   VAR_OUTPUT
      q_UDT_Status { ExternalAccessible := 'False'; ExternalVisible := 'False'; ExternalWritable := 'False'} : "UDT_SecurityCageStatus";   // Status
      qx_StartStopButtonLamp { ExternalAccessible := 'False'; ExternalVisible := 'False'; ExternalWritable := 'False'} : Bool;   // Start stop lamp button
      qx_DirectionButtonLamp { ExternalAccessible := 'False'; ExternalVisible := 'False'; ExternalWritable := 'False'} : Bool;   // Direction lamp button
      qx_ReverseDirection { ExternalAccessible := 'False'; ExternalVisible := 'False'; ExternalWritable := 'False'} : Bool;   // Signal to the system to change line direction
   END_VAR

   VAR_IN_OUT
      iq_UDT_SystemControlCommand : "UDT_SystemControlCommand";   // HMI system control structure
      iq_UDT_EquipmentControl : "UDT_EquipmentControl";   // Equipment control structure
   END_VAR

   VAR
      R_TRIG_StartStopButton {InstructionName := 'R_TRIG'; LibVersion := '1.0'; ExternalAccessible := 'False'; ExternalVisible := 'False'; ExternalWritable := 'False'; S7_SetPoint := 'False'} : R_TRIG;   // Rising edge trigger of start stop button
      R_TRIG_DirectionButton {InstructionName := 'R_TRIG'; LibVersion := '1.0'; ExternalAccessible := 'False'; ExternalVisible := 'False'; ExternalWritable := 'False'; S7_SetPoint := 'False'} : R_TRIG;   // Rising edge trigger of direction button
      sx_StartStopButtonLamp { ExternalAccessible := 'False'; ExternalVisible := 'False'; ExternalWritable := 'False'} : Bool;   // Start stop lamp button
      sx_DirectionButtonLamp { ExternalAccessible := 'False'; ExternalVisible := 'False'; ExternalWritable := 'False'} : Bool;   // Direction lamp button
      sx_Infeed { ExternalAccessible := 'False'; ExternalVisible := 'False'; ExternalWritable := 'False'} : Bool := TRUE;   // Infeed mode
      sx_Outfeed { ExternalAccessible := 'False'; ExternalVisible := 'False'; ExternalWritable := 'False'} : Bool;   // Outfeed mode
   END_VAR


BEGIN
	(*
	----------------------------------------------------------------------------------------
	|                                                                                      |
	|  Copyright  2023             Fortna Europe BV                                        |
	|  All Rights Reserved         Netherlands                                             |
	|                                                                                      |
	|                                                                                      |
	----------------------------------------------------------------------------------------

	Version history:
	Date        | Version   | Author       | Remark
	----------------------------------------------------------------------------------------
	23/11/2022  | 1.0       | S. Nikodem   | Release TIA 17 | DHL Munich 2023
	13/03/2024  | 1.1       | S. Nieswiec  | Added to new Baseline
	*)

	REGION 1 - Triggers

	    #R_TRIG_StartStopButton(CLK := #ix_StartStopButton);
	    #R_TRIG_DirectionButton(CLK := #ix_DirectionButton);

	END_REGION

	REGION 2 - Start Stop System

	    //If system is running then stop the system
	    IF #iq_UDT_EquipmentControl.Command.AutomaticOn AND #R_TRIG_StartStopButton.Q THEN

	        #iq_UDT_SystemControlCommand.Stop := True;

	    END_IF;

	    //If system is stopped then start the system
	    IF NOT #iq_UDT_EquipmentControl.Command.AutomaticOn AND #R_TRIG_StartStopButton.Q THEN

	        #iq_UDT_SystemControlCommand.Start := True;

	    END_IF;

	END_REGION

	REGION 3 - Mode

	    //Select mode
	    // The mode can be only changed when the line is stopped

	    IF NOT #iq_UDT_EquipmentControl.Command.AutomaticOn AND #R_TRIG_DirectionButton.Q THEN

	        #sx_Infeed := NOT #sx_Infeed;
	        #sx_Outfeed := NOT #sx_Outfeed;


	    END_IF;

	END_REGION

	REGION 4 - Lamp operation

	    //When the selected direction is infeed (from ground floor to security cage) the button will be solid on
	    //When the selected direction is outfeed (from the security cage to ground floor) THEN the button will be flashing at 1Hz.
	    #sx_DirectionButtonLamp := #sx_Infeed OR (#sx_Outfeed AND "mx_Clock_1Hz");


	    //When system is running then lamp will be solid on.
	    #sx_StartStopButtonLamp := #iq_UDT_EquipmentControl.Command.AutomaticOn;

	END_REGION

	REGION 5 - Status

	    #q_UDT_Status.InfeedMode := #sx_Infeed;
	    #q_UDT_Status.OutfeedMode := #sx_Outfeed;

	END_REGION

	REGION 6 - Write outputs
	    #qx_ReverseDirection := #sx_Outfeed;
	    #qx_StartStopButtonLamp := #sx_StartStopButtonLamp;
	    #qx_DirectionButtonLamp := #sx_DirectionButtonLamp;

	END_REGION

END_FUNCTION_BLOCK

FUNCTION_BLOCK "FB_RetractableRoller"
{ S7_Optimized_Access := 'TRUE' }
VERSION : 0.1
// ATTRIBUTES
// AUTO_NUMBER = True
// BLOCK_NUMBER = 100
// END_ATTRIBUTES
   VAR_INPUT
      ix_RollerError { ExternalAccessible := 'False'; ExternalVisible := 'False'; ExternalWritable := 'False'} : Bool;   // Error from roller
      ix_RollerAtHome { ExternalAccessible := 'False'; ExternalVisible := 'False'; ExternalWritable := 'False'} : Bool;   // Roller at home position
      ix_Button { ExternalAccessible := 'False'; ExternalVisible := 'False'; ExternalWritable := 'False'} : Bool;   // Switching on/off the magnet
      ix_DirectionConfig { ExternalAccessible := 'False'; ExternalVisible := 'False'; ExternalWritable := 'False'} : Bool;   // Change the direction
   END_VAR

   VAR_OUTPUT
      qx_RollerCW { ExternalAccessible := 'False'; ExternalVisible := 'False'; ExternalWritable := 'False'} : Bool;   // Forward direction
      qx_RollerCCW { ExternalAccessible := 'False'; ExternalVisible := 'False'; ExternalWritable := 'False'} : Bool;   // Revers direction
      qx_RollerRun { ExternalAccessible := 'False'; ExternalVisible := 'False'; ExternalWritable := 'False'} : Bool;   // Run Roller
      qx_Magnet { ExternalAccessible := 'False'; ExternalVisible := 'False'; ExternalWritable := 'False'} : Bool;   // On/Off Magnet
      qx_ConveyorInDieBack { ExternalAccessible := 'False'; ExternalVisible := 'False'; ExternalWritable := 'False'} : Bool;   // Active DieBack mode
      q_UDT_HMIStatus { ExternalAccessible := 'False'; ExternalVisible := 'False'; ExternalWritable := 'False'} : "UDT_RetractrableRoller_Status";   // HMI status structure
   END_VAR

   VAR_IN_OUT
      iq_UDT_ConveyorInterface : "UDT_ConveyorInterface";   // Interface structure
   END_VAR

   VAR
      s_UDT_HMI_Status { ExternalAccessible := 'False'; ExternalVisible := 'False'; ExternalWritable := 'False'; S7_SetPoint := 'False'} : "UDT_RetractrableRoller_Status";   // RetractrableRoller structure
      sx_RollerRun { ExternalAccessible := 'False'; ExternalVisible := 'False'; ExternalWritable := 'False'} : Bool;   // Roller is active
      sx_RollerCW { ExternalAccessible := 'False'; ExternalVisible := 'False'; ExternalWritable := 'False'} : Bool;   // Roller is in forward mode
      sx_RollerCCW { ExternalAccessible := 'False'; ExternalVisible := 'False'; ExternalWritable := 'False'} : Bool;   // Roller is in revers mode
      sx_Magnet { ExternalAccessible := 'False'; ExternalVisible := 'False'; ExternalWritable := 'False'} : Bool;   // Magnet is active
      sx_ConveyorInDieBack { ExternalAccessible := 'False'; ExternalVisible := 'False'; ExternalWritable := 'False'} : Bool;   // Dieback mode active
      s_UDT_CommonStatus { ExternalAccessible := 'False'; ExternalVisible := 'False'; ExternalWritable := 'False'; S7_SetPoint := 'False'} : "UDT_CommonStatus";   // Common status structure
      s_UDT_CommonStatusOld { ExternalAccessible := 'False'; ExternalVisible := 'False'; ExternalWritable := 'False'; S7_SetPoint := 'False'} : "UDT_CommonStatus";   // Common status structure
   END_VAR


BEGIN
	(*
	----------------------------------------------------------------------------------------
	|                                                                                      |
	|  Copyright  2023             FORTNA Europe BV                                        |
	|  All Rights Reserved         Netherlands                                             |
	|                                                                                      |
	----------------------------------------------------------------------------------------
	Version history:
	Date        | Version   | Author       | Remark
	----------------------------------------------------------------------------------------
	05/05/2023  | 1.0       | M. Diebel   | Release TIA 17 | DHL Munich 2023
	13/03/2024  | 1.1       | S. Nieswiec  | Added to new Baseline
	*)

	REGION 1 - Magnet handling

	    //Keep true the magnet output when the Proxy detects roller and the button is not pressed
	    #sx_Magnet := #ix_RollerAtHome AND NOT #ix_Button;

	END_REGION

	REGION 2 - Roller handling

	    // Run rollers
	    #sx_RollerRun := #ix_RollerAtHome AND (#iq_UDT_ConveyorInterface.RunFwd OR #iq_UDT_ConveyorInterface.RunRvs);

	    // Roller direction
	    IF NOT #ix_DirectionConfig
	    THEN

	        // Run rollers in forward mode
	        #sx_RollerCW := #ix_RollerAtHome AND #iq_UDT_ConveyorInterface.RunFwd AND NOT #iq_UDT_ConveyorInterface.RunRvs;

	        // Run rollers in revers mode
	        #sx_RollerCCW := #ix_RollerAtHome AND #iq_UDT_ConveyorInterface.RunRvs AND NOT #iq_UDT_ConveyorInterface.RunFwd;

	    ELSE

	        // Run rollers in forward mode
	        #sx_RollerCW := #ix_RollerAtHome AND #iq_UDT_ConveyorInterface.RunRvs AND NOT #iq_UDT_ConveyorInterface.RunFwd;

	        // Run rollers in revers mode
	        #sx_RollerCCW := #ix_RollerAtHome AND #iq_UDT_ConveyorInterface.RunFwd AND NOT #iq_UDT_ConveyorInterface.RunRvs;

	    END_IF;

	    // DieBack mode for Conveyor when roller is not at home position
	    #sx_ConveyorInDieBack := NOT #ix_RollerAtHome;

	    // Rollers is not in home position
	    #s_UDT_HMI_Status.Specific.NoHomePosition := NOT #ix_RollerAtHome;

	    // Roller reports an error
	    #s_UDT_HMI_Status.Specific.RollerError := #ix_RollerError;

	END_REGION

	REGION 3 - Status

	    //Error
	    #s_UDT_CommonStatus.Error := #s_UDT_HMI_Status.Specific.NoHomePosition;

	    //Running
	    #s_UDT_CommonStatus.Running := #sx_RollerRun AND NOT #s_UDT_HMI_Status.Specific.NoHomePosition;

	    //Stopped
	    #s_UDT_CommonStatus.Stopped := NOT #sx_RollerRun AND NOT #s_UDT_HMI_Status.Specific.NoHomePosition;

	    IF #s_UDT_CommonStatusOld <> #s_UDT_CommonStatus
	    THEN
	        // HMI status initialization
	        #s_UDT_HMI_Status.Status := 0;

	        IF #s_UDT_CommonStatus.Error
	        THEN
	            #s_UDT_HMI_Status.Status := "DB_HMIStatusConfiguration".Error;
	        END_IF;

	        IF #s_UDT_CommonStatus.Running
	        THEN
	            #s_UDT_HMI_Status.Status := "DB_HMIStatusConfiguration".Running;
	        END_IF;

	        IF #s_UDT_CommonStatus.Stopped
	        THEN
	            #s_UDT_HMI_Status.Status := "DB_HMIStatusConfiguration".Stopped;
	        END_IF;

	        #s_UDT_CommonStatusOld := #s_UDT_CommonStatus;

	    END_IF;

	END_REGION

	REGION 4 - Update outputs

	    #q_UDT_HMIStatus := #s_UDT_HMI_Status;
	    #qx_RollerCW := #sx_RollerCW;
	    #qx_RollerCCW := #sx_RollerCCW;
	    #qx_RollerRun := #sx_RollerRun;
	    #qx_Magnet := #sx_Magnet;
	    #qx_ConveyorInDieBack := #sx_ConveyorInDieBack;

	END_REGION
END_FUNCTION_BLOCK

FUNCTION_BLOCK "FB_Outfeed2States"
{ S7_Optimized_Access := 'TRUE' }
VERSION : 2.0
// ATTRIBUTES
// AUTO_NUMBER = True
// BLOCK_NUMBER = 99
// END_ATTRIBUTES
   VAR_INPUT
      i_UDT_ChuteConfiguration { ExternalAccessible := 'False'; ExternalVisible := 'False'; ExternalWritable := 'False'} : "UDT_Outfeed2StatesConfiguration";   // Chute Configuration structure
      i_UDT_AssociatedConveyorStatus { ExternalAccessible := 'False'; ExternalVisible := 'False'; ExternalWritable := 'False'} : "UDT_CommonStatus";   // Conveyor status
      ix_CapacityControlActive { ExternalAccessible := 'False'; ExternalVisible := 'False'; ExternalWritable := 'False'} : Bool;   // Chute capacity control is full
      ix_Enable { ExternalAccessible := 'False'; ExternalVisible := 'False'; ExternalWritable := 'False'} : Bool;   // TRUE when chute funcktion is enable
      ix_ConditionFull { ExternalAccessible := 'False'; ExternalVisible := 'False'; ExternalWritable := 'False'} : Bool;   // TRUE when Chute Full contidion is not blocked
      ix_ConditionHalfFull { ExternalAccessible := 'False'; ExternalVisible := 'False'; ExternalWritable := 'False'} : Bool;   // TRUE when Chute Half Full condition is not blocked
      ix_Disabled { ExternalAccessible := 'False'; ExternalVisible := 'False'; ExternalWritable := 'False'} : Bool;   // TRUE when chute is disabled
      ix_HardwareOk { ExternalAccessible := 'False'; ExternalVisible := 'False'; ExternalWritable := 'False'} : Bool;   // TRUE when chute hardware is Ok
      iudi_DelayHardwareOK { ExternalAccessible := 'False'; ExternalVisible := 'False'; ExternalWritable := 'False'} : UDInt;   // Time to delay for hardware ok signal
   END_VAR

   VAR_OUTPUT
      qx_Lamp { ExternalAccessible := 'False'; ExternalVisible := 'False'; ExternalWritable := 'False'} : Bool;   // Output Chute Lamp half full/ full
      q_UDT_HMIStatus { ExternalAccessible := 'False'; ExternalVisible := 'False'; ExternalWritable := 'False'} : "UDT_Outfeed2StatesStatus";   // HMI chute status structure
      q_UDT_Status { ExternalAccessible := 'False'; ExternalVisible := 'False'; ExternalWritable := 'False'} : "UDT_CommonStatus";   // Common chute status structure
   END_VAR

   VAR_IN_OUT
      iq_UDT_EquipmentControl : "UDT_EquipmentControl";   // Equipment control structure
      iq_ChuteExternalHandshake : "UDT_ConveyorHandshake";   // Upstream handshake structure
      iq_UDT_ConveyorHandshake : "UDT_ConveyorHandshake";
      iq_UDT_Statistics : "UDT_Outfeed2StatesStatistics";   // Statistics structure
   END_VAR

   VAR
      s_UDT_HMIStatus { ExternalAccessible := 'False'; ExternalVisible := 'False'; ExternalWritable := 'False'; S7_SetPoint := 'False'} : "UDT_Outfeed2StatesStatus";   // HMI status structure
      s_UDT_CommonStatus { ExternalAccessible := 'False'; ExternalVisible := 'False'; ExternalWritable := 'False'; S7_SetPoint := 'False'} : "UDT_CommonStatus";   // Common status structure
      s_UDT_CommonStatusOld { ExternalAccessible := 'False'; ExternalVisible := 'False'; ExternalWritable := 'False'; S7_SetPoint := 'False'} : "UDT_CommonStatus";   // Auxiliary status structure
      s_FB_HardwareOk { ExternalAccessible := 'False'; ExternalVisible := 'False'; ExternalWritable := 'False'; S7_SetPoint := 'False'} : "FB_TimerOnOffDelay";   // Timer on/off delay for hardware ok signal
      s_FB_ChuteHalfFullDetectionDelay { ExternalAccessible := 'False'; ExternalVisible := 'False'; ExternalWritable := 'False'; S7_SetPoint := 'False'} : "FB_TimerOnOffDelay";   // Timer on/off delay for chute half  full detection
      s_FB_ChuteFullDetectionDelay { ExternalAccessible := 'False'; ExternalVisible := 'False'; ExternalWritable := 'False'; S7_SetPoint := 'False'} : "FB_TimerOnOffDelay";   // Timer on/off delay for chute full detection
      s_R_TRIG_HalfFull {InstructionName := 'R_TRIG'; LibVersion := '1.0'; ExternalAccessible := 'False'; ExternalVisible := 'False'; ExternalWritable := 'False'; S7_SetPoint := 'False'} : R_TRIG;   // Rising edge trigger on chute half full signal
      s_R_TRIG_Disabled {InstructionName := 'R_TRIG'; LibVersion := '1.0'; ExternalAccessible := 'False'; ExternalVisible := 'False'; ExternalWritable := 'False'; S7_SetPoint := 'False'} : R_TRIG;   // Rising edge trigger on chute disabled signal
      s_R_TRIG_ChuteFull {InstructionName := 'R_TRIG'; LibVersion := '1.0'; ExternalAccessible := 'False'; ExternalVisible := 'False'; ExternalWritable := 'False'; S7_SetPoint := 'False'} : R_TRIG;   // Rising edge trigger on chute full signal
      s_F_TRIG_UpdateStatus {InstructionName := 'F_TRIG'; LibVersion := '1.0'; ExternalAccessible := 'False'; ExternalVisible := 'False'; ExternalWritable := 'False'; S7_SetPoint := 'False'} : F_TRIG;   // Falling edge trigger on status change
      sx_Full { ExternalAccessible := 'False'; ExternalVisible := 'False'; ExternalWritable := 'False'} : Bool;   // Full status
      sx_HalfFull { ExternalAccessible := 'False'; ExternalVisible := 'False'; ExternalWritable := 'False'} : Bool;   // Half full status
   END_VAR


BEGIN
	(*
	----------------------------------------------------------------------------------------
	|                                                                                      |
	|  Copyright  2023             FORTNA Europe BV                                        |
	|  All Rights Reserved         Netherlands                                             |
	|                                                                                      |
	----------------------------------------------------------------------------------------

	Version history:
	Date        | Version   | Author            | Remark
	----------------------------------------------------------------------------------------
	 01/03/2023 | 1.0       | R. Golonka        | Release V17 | DHL Munich
	 05/09/2023 | 1.1       | S.Theocharis      | remove the reset of restart required
	 05/09/2023 | 1.2       | M.Diebel          | Initilization, s_UDT_CommonStatus.Stopped set on true
	 06/09/2023 | 1.3       | M.Diebel          | Rewrite reset energy save from external handshake to conveyor handshake
	 12/09/2023 | 2.0       | M.Diebel          | Set status "stopped" when chute is disable
	 13/03/2024 | 2.1       | S. Nieswiec       | Added to new Baseline


	 *)


	REGION 1 - Inicialization
	    //Reset HMI status and Common status and exit
	    IF NOT #ix_Enable THEN
	        #s_UDT_HMIStatus.Specific.ChuteFull := 0;
	        #s_UDT_HMIStatus.Specific.ChuteHalfFull := 0;
	        #s_UDT_HMIStatus.Specific.ChuteDisabled := 0;
	        #s_UDT_CommonStatus.SafetyStop := 0;
	        #s_UDT_CommonStatus.AutoON := 0;
	        #s_UDT_CommonStatus.Stopped := TRUE;
	        #s_UDT_HMIStatus.Status := "DB_HMIStatusConfiguration".Stopped;
	        #q_UDT_HMIStatus := #s_UDT_HMIStatus;
	        #q_UDT_Status := #s_UDT_CommonStatus;
	        #iq_UDT_EquipmentControl.Report := #s_UDT_CommonStatus;
	        #qx_Lamp := 0;
	        #iq_UDT_ConveyorHandshake.RTS := 0;
	        #iq_ChuteExternalHandshake.RTR := 0;

	        RETURN;
	    END_IF;
	END_REGION

	REGION 2 - Timers

	    // Chute full detection timer
	    #s_FB_ChuteFullDetectionDelay(iudi_OnDelayTime := #i_UDT_ChuteConfiguration.FullDetectionTime,
	                                  iudi_OffDelayTime := #i_UDT_ChuteConfiguration.FullReleaseTime,
	                                  ix_SignalToDelay := NOT #ix_ConditionFull,
	                                  qx_DelayedSignal => #sx_Full);

	    // Chute half full detection timer
	    #s_FB_ChuteHalfFullDetectionDelay(iudi_OnDelayTime := #i_UDT_ChuteConfiguration.HalfFullDetectionTime,
	                                      iudi_OffDelayTime := #i_UDT_ChuteConfiguration.HalfFullReleaseTime,
	                                      ix_SignalToDelay := NOT #ix_ConditionHalfFull,
	                                      qx_DelayedSignal => #sx_HalfFull);

	    // Hardware ok signal delay
	    #s_FB_HardwareOk(iudi_OnDelayTime := #iudi_DelayHardwareOK,
	                     ix_SignalToDelay := #ix_HardwareOk);


	END_REGION

	REGION 3 - Stop upstream conveyor

	    // Stop upstream conveyor when chute is full or disabled
	    #iq_ChuteExternalHandshake.RTR := NOT #sx_Full AND NOT #ix_CapacityControlActive AND NOT #ix_Disabled AND #s_FB_HardwareOk.qx_DelayedSignal AND #iq_UDT_EquipmentControl.Report.AutoON;

	END_REGION

	REGION 4 - Start next conveyor

	    // Start conveyor when upstream conveyor is running
	    #iq_UDT_ConveyorHandshake.RTS := #iq_ChuteExternalHandshake.RTR;
	    #iq_UDT_ConveyorHandshake.ResetEnergySave := #iq_ChuteExternalHandshake.ResetEnergySave;
	END_REGION


	REGION 5 - Update output

	    // Update the outputs
	    #qx_Lamp := (#sx_Full OR (#sx_HalfFull AND "DB_Memory".Clock_1Hz));

	END_REGION

	REGION 6 - Status

	    // Update chute full specific status
	    #s_UDT_HMIStatus.Specific.ChuteFull := #sx_Full AND #s_FB_HardwareOk.qx_DelayedSignal;

	    // Update chute half full specific status
	    #s_UDT_HMIStatus.Specific.ChuteHalfFull := #sx_HalfFull AND #s_FB_HardwareOk.qx_DelayedSignal;

	    //Update chute disabled specific status
	    #s_UDT_HMIStatus.Specific.ChuteDisabled := #ix_Disabled AND #s_FB_HardwareOk.qx_DelayedSignal;


	    // Update common safety stop
	    #s_UDT_CommonStatus.SafetyStop := #i_UDT_AssociatedConveyorStatus.SafetyStop;

	    // Update common automatic on
	    #s_UDT_CommonStatus.AutoON := #i_UDT_AssociatedConveyorStatus.AutoON;

	    // Update common stopped
	    #s_UDT_CommonStatus.Stopped := #i_UDT_AssociatedConveyorStatus.Stopped;


	    // Update HMI status number for chute disabled
	    IF #s_UDT_HMIStatus.Specific.ChuteDisabled AND NOT #s_UDT_CommonStatus.SafetyStop
	    THEN
	        #s_UDT_HMIStatus.Status := "DB_HMIStatusConfiguration".DisableByManagement;
	    END_IF;

	    // Update HMI status number for chute half full
	    IF #s_UDT_HMIStatus.Specific.ChuteHalfFull AND NOT #s_UDT_CommonStatus.SafetyStop
	    THEN
	        #s_UDT_HMIStatus.Status := "DB_HMIStatusConfiguration".ChuteHalfFull;
	    END_IF;

	    // Update HMI status number for chute full
	    IF #s_UDT_HMIStatus.Specific.ChuteFull AND NOT #s_UDT_CommonStatus.SafetyStop
	    THEN
	        #s_UDT_HMIStatus.Status := "DB_HMIStatusConfiguration".ChuteFull;
	    END_IF;


	    // Collecting F_TRIG on chute full, chute half full or chute disabled status to update common status
	    #s_F_TRIG_UpdateStatus(CLK := #s_UDT_HMIStatus.Specific.ChuteFull
	                           OR #s_UDT_HMIStatus.Specific.ChuteDisabled
	                           OR #s_UDT_HMIStatus.Specific.ChuteHalfFull);

	    // HMI status number calculation
	    IF #s_UDT_CommonStatusOld <> #s_UDT_CommonStatus OR #s_F_TRIG_UpdateStatus.Q
	    THEN

	        // Update auto on status number
	        IF #s_UDT_CommonStatus.AutoON
	        THEN
	            #s_UDT_HMIStatus.Status := "DB_HMIStatusConfiguration".AutoON;

	        END_IF;

	        IF #s_UDT_CommonStatus.Stopped
	        THEN
	            #s_UDT_HMIStatus.Status := "DB_HMIStatusConfiguration".Stopped;

	        END_IF;

	        IF #s_UDT_CommonStatus.SafetyStop
	        THEN
	            #s_UDT_HMIStatus.Status := "DB_HMIStatusConfiguration".SafetyStop;

	        END_IF;

	        // Copy common status structure to the old common status structure
	        #s_UDT_CommonStatusOld := #s_UDT_CommonStatus;
	        #q_UDT_Status := #s_UDT_CommonStatus;

	    END_IF;

	    #q_UDT_HMIStatus := #s_UDT_HMIStatus;

	END_REGION

	REGION 7 - Statistics

	    // Chute full R_TRIG for statistics purpose
	    #s_R_TRIG_ChuteFull(CLK := #s_UDT_HMIStatus.Specific.ChuteFull);

	    // Chute full statistics
	    IF #s_UDT_HMIStatus.Specific.ChuteFull
	        OR #iq_UDT_EquipmentControl.Command.ResetData
	    THEN
	        "FC_Statistics"(ix_Reset := #iq_UDT_EquipmentControl.Command.ResetData,
	                        ix_Activate := #s_UDT_HMIStatus.Specific.ChuteFull,
	                        ix_RTrigActivate := #s_R_TRIG_ChuteFull.Q,
	                        iqUDT_Statistics := #iq_UDT_Statistics.ChuteFull);

	    END_IF;

	    // Chute disabled R_TRIG for statistics purpose
	    #s_R_TRIG_Disabled(CLK := #s_UDT_HMIStatus.Specific.ChuteDisabled);

	    // Chute disabled statistics
	    IF #s_UDT_HMIStatus.Specific.ChuteDisabled
	        OR #iq_UDT_EquipmentControl.Command.ResetData
	    THEN
	        "FC_Statistics"(ix_Reset := #iq_UDT_EquipmentControl.Command.ResetData,
	                        ix_Activate := #s_UDT_HMIStatus.Specific.ChuteDisabled,
	                        ix_RTrigActivate := #s_R_TRIG_Disabled.Q,
	                        iqUDT_Statistics := #iq_UDT_Statistics.ChuteDisabled);

	    END_IF;

	    // Chute half full R_TRIG for statistics purpose
	    #s_R_TRIG_HalfFull(CLK := #s_UDT_HMIStatus.Specific.ChuteHalfFull);

	    // Chute half full statistics
	    IF #s_UDT_HMIStatus.Specific.ChuteHalfFull
	        OR #iq_UDT_EquipmentControl.Command.ResetData
	    THEN

	        "FC_Statistics"(ix_Reset := #iq_UDT_EquipmentControl.Command.ResetData,
	                        ix_Activate := #s_UDT_HMIStatus.Specific.ChuteHalfFull,
	                        ix_RTrigActivate := #s_R_TRIG_HalfFull.Q,
	                        iqUDT_Statistics := #iq_UDT_Statistics.ChuteHalfFull);

	    END_IF;

	END_REGION

	REGION 8 - Equipment Report

	    "FC_EquipmentReport"(iUDT_Status := #s_UDT_CommonStatus,
	                         iqUDT_Control := #iq_UDT_EquipmentControl);

	END_REGION
END_FUNCTION_BLOCK

FUNCTION_BLOCK "FB_InchingBulkV2"
{ S7_Optimized_Access := 'TRUE' }
VERSION : 0.1
// ATTRIBUTES
// AUTO_NUMBER = True
// BLOCK_NUMBER = 97
// END_ATTRIBUTES
   VAR_INPUT
      ix_PECUp { ExternalAccessible := 'False'; ExternalVisible := 'False'; ExternalWritable := 'False'} : Bool;   // PEC Sum signal from upstream conveyor
      ix_LongParcelDetection { ExternalAccessible := 'False'; ExternalVisible := 'False'; ExternalWritable := 'False'} : Bool;   // Long parcel detection PEC's
      ix_InchingActive { ExternalAccessible := 'False'; ExternalVisible := 'False'; ExternalWritable := 'False'} : Bool;   // If TRUE inching is activate
      ix_InchingLineHealthy { ExternalAccessible := 'False'; ExternalVisible := 'False'; ExternalWritable := 'False'} : Bool;
      ix_ClearCommand { ExternalAccessible := 'False'; ExternalVisible := 'False'; ExternalWritable := 'False'} : Bool;   // Command to clear full status
      ix_DownstreamFull { ExternalAccessible := 'False'; ExternalVisible := 'False'; ExternalWritable := 'False'} : Bool;   // TRUE if downstream conveyors are full
      ii_OnDelayGap { ExternalAccessible := 'False'; ExternalVisible := 'False'; ExternalWritable := 'False'} : DInt;   // Distance to conveyor release [mm]
      ii_InchingGap { ExternalAccessible := 'False'; ExternalVisible := 'False'; ExternalWritable := 'False'} : DInt;   // Inching distance [mm]
      ii_Displacement_Upstream { ExternalAccessible := 'False'; ExternalVisible := 'False'; ExternalWritable := 'False'} : Int;   // Upstream conveyor displacement
      ii_Displacement { ExternalAccessible := 'False'; ExternalVisible := 'False'; ExternalWritable := 'False'} : Int;   // Inching conveyor displacement
      iudt_ConveyorInterface { ExternalAccessible := 'False'; ExternalVisible := 'False'; ExternalWritable := 'False'} : "UDT_ConveyorInterface";
   END_VAR

   VAR_OUTPUT
      qx_ExternalRequestHold { ExternalAccessible := 'False'; ExternalVisible := 'False'; ExternalWritable := 'False'} : Bool;   // External output to request conveyor hold
      qx_Full { ExternalAccessible := 'False'; ExternalVisible := 'False'; ExternalWritable := 'False'} : Bool;   // Inching conveyor is full status
   END_VAR

   VAR
      s_FB_TimerOnOffDelay_LongParcelDetection { ExternalAccessible := 'False'; ExternalVisible := 'False'; ExternalWritable := 'False'; S7_SetPoint := 'False'} : "FB_TimerOnOffDelay";
      F_TRIG_PECEoSUp {InstructionName := 'F_TRIG'; LibVersion := '1.0'; ExternalAccessible := 'False'; ExternalVisible := 'False'; ExternalWritable := 'False'; S7_SetPoint := 'False'} : F_TRIG;   // Falling edge trigger PEC EoS
      si_ActualInchingGap { ExternalAccessible := 'False'; ExternalVisible := 'False'; ExternalWritable := 'False'} : Int;   // Distance to request hold
      si_ActualOnGap { ExternalAccessible := 'False'; ExternalVisible := 'False'; ExternalWritable := 'False'} : Int;   // Distance to conveyor release
      sx_StartRelease { ExternalAccessible := 'False'; ExternalVisible := 'False'; ExternalWritable := 'False'} : Bool;   // Conveyor release
      sx_ConveyorFull { ExternalAccessible := 'False'; ExternalVisible := 'False'; ExternalWritable := 'False'} : Bool;
      s_Status { ExternalAccessible := 'False'; ExternalVisible := 'False'; ExternalWritable := 'False'; S7_SetPoint := 'False'} : "UDT_InchingStatus";
      s_StatusOld { ExternalAccessible := 'False'; ExternalVisible := 'False'; ExternalWritable := 'False'; S7_SetPoint := 'False'} : "UDT_InchingStatus";
      sx_InchingActive { ExternalAccessible := 'False'; ExternalVisible := 'False'; ExternalWritable := 'False'} : Bool;
   END_VAR


BEGIN
	(*
	----------------------------------------------------------------------------------------
	|                                                                                      |
	|  Copyright  2019             MHS                                                     |
	|  All Rights Rese9ved         Larenweg 90                                             |
	|                              5234 KC 's-Hertogenbosch,                               |
	|                              Netherlands                                             |
	|                                                                                      |
	----------------------------------------------------------------------------------------

	Version history:
	Date        | Version   | Author        | Remark
	----------------------------------------------------------------------------------------
	01/04/2021 | 1.0       | M.Kocot      | first release TIA 16
	08/04/2021 | 1.1       | H.Rutkwoski  | Added status full
	14/08/2021 | 1.2       | M. Jager     | Reset sx_full when inching is not active
	26/07/2023 | 1.3       | S.Nikodem    | Absolut displacement value
	13/09/2023 | 1.4       | M.Diebel     | Activate inching if PEC is clear
	14/09/2023 | 1.5       | M.Diebel     | Hold line when downstream conveyors are full
	06/02/2024 | 1.6       | L.Klar       | Long parcel detection
	13/03/2024 | 1.7       | S. Nieswiec  | Changed name to V2
	*)

	REGION 1 - Triggers

	    // Falling edge trigger PEC EoS.
	    #F_TRIG_PECEoSUp(CLK := #ix_PECUp);

	END_REGION

	REGION 2 - TTimers

	    #s_FB_TimerOnOffDelay_LongParcelDetection(iudi_OffDelayTime := 100,
	                                              ix_SignalToDelay := #ix_LongParcelDetection);

	END_REGION

	REGION 3 - Inching
	    // Statement section REGION

	    //Activate inching if PEC is clear
	    #sx_InchingActive := #ix_InchingActive AND (#sx_InchingActive OR #ix_PECUp);



	    IF ((#F_TRIG_PECEoSUp.Q OR NOT #s_FB_TimerOnOffDelay_LongParcelDetection.qx_DelayedSignal) AND #sx_InchingActive)
	        // OR( RisingeEdge of Ix_InchigActive AND NOT IX_PECup )
	    THEN
	        #si_ActualOnGap := DINT_TO_INT(#ii_OnDelayGap / 10);
	        #si_ActualInchingGap := DINT_TO_INT(#ii_InchingGap / 10);

	    END_IF;

	    IF #si_ActualOnGap > 0 THEN

	        #si_ActualOnGap := #si_ActualOnGap - ABS(#ii_Displacement_Upstream);

	    END_IF;

	    IF #ix_PECUp AND #si_ActualInchingGap > 0 THEN
	        #si_ActualInchingGap := #si_ActualInchingGap - ABS(#ii_Displacement);
	    END_IF;

	    IF #si_ActualOnGap <= 0
	        //  OR #sx_StartRelease
	    THEN
	        #sx_StartRelease := TRUE;
	    END_IF;

	    IF (#si_ActualInchingGap <= 0)
	    THEN
	        #sx_StartRelease := FALSE;
	    END_IF;

	    #qx_ExternalRequestHold := (((NOT #sx_StartRelease OR NOT #ix_InchingLineHealthy) OR #ix_DownstreamFull) AND #sx_InchingActive);

	END_REGION

	REGION 4 - Internal status - conveyor full

	    // Set conveyor status to full when:
	    IF #sx_InchingActive                     // inching is active
	        AND #ix_DownstreamFull               // downstream is full
	        AND NOT #ix_ClearCommand             // there is no clear command active
	    THEN
	        #sx_ConveyorFull := TRUE;
	    END_IF;

	    // Set conveyor status to NOT full when:
	    IF (#sx_InchingActive                   // Inching is active
	        AND #ix_ClearCommand                // clear command is active
	        AND NOT #ix_DownstreamFull)         // downstream is NOT full)
	        OR NOT #sx_InchingActive            // OR Inching isnt active
	    THEN
	        #sx_ConveyorFull := FALSE;
	    END_IF;

	END_REGION

	REGION 5 - Status

	    // Convsyor is full status
	    #s_Status.Full := #sx_ConveyorFull;

	    #s_Status.Active := #sx_InchingActive;

	    // Status update on change.
	    IF #s_StatusOld <> #s_Status
	    THEN
	        #qx_Full := #s_Status.Full;
	        #s_StatusOld := #s_Status;
	    END_IF;

	END_REGION
END_FUNCTION_BLOCK

FUNCTION_BLOCK "FB_SNCY_Infeed"
{ S7_Optimized_Access := 'TRUE' }
VERSION : 0.1
// ATTRIBUTES
// AUTO_NUMBER = True
// BLOCK_NUMBER = 242
// END_ATTRIBUTES
   VAR_INPUT
      ix_KneeButton { ExternalAccessible := 'False'; ExternalVisible := 'False'; ExternalWritable := 'False'} : Bool;   // Signal from knee button
      ix_ResetButton { ExternalAccessible := 'False'; ExternalVisible := 'False'; ExternalWritable := 'False'} : Bool;   // Signal from reset button
      ix_PEC_EoS { ExternalAccessible := 'False'; ExternalVisible := 'False'; ExternalWritable := 'False'} : Bool;   // Sensor at end of conveyor
      i_UDT_PECUpdateConfiguration { ExternalAccessible := 'False'; ExternalVisible := 'False'; ExternalWritable := 'False'} : "UDT_PECUpdateConfiguration";   // PEC update configuration
      idtl_ActualTime {InstructionName := 'DTL'; LibVersion := '1.0'; ExternalAccessible := 'False'; ExternalVisible := 'False'; ExternalWritable := 'False'} : DTL;   // Actual date and time in DTL
   END_VAR

   VAR_OUTPUT
      qx_ConveyorHold { ExternalAccessible := 'False'; ExternalVisible := 'False'; ExternalWritable := 'False'} : Bool;   // Hold command for conveyor
      qx_WhiteLamp { ExternalAccessible := 'False'; ExternalVisible := 'False'; ExternalWritable := 'False'} : Bool;   // White signal lamp
      qx_BlueLamp { ExternalAccessible := 'False'; ExternalVisible := 'False'; ExternalWritable := 'False'} : Bool;   // Blue signal lamp
   END_VAR

   VAR_IN_OUT
      iqa_TrackingData : Array[*] of Int;   // Conveyor tracking data
      iq_UDT_FifoHeaderMFCMessage : "UDT_FifoHeader";   // FIFO header of generated messages
      iqs_FifoDataMFCMessage : Array[*] of "UDT_MessageV2";   // FIFO data Buffer of generated messages
      iqdi_MessageSequenceNumber { ExternalAccessible := 'False'; ExternalVisible := 'False'; ExternalWritable := 'False'} : Int;   // MFC Sort - Message number
      iqs_MFCNewObjectID : String;   // New Object ID number received from MFC
      is_MFCRejectObjectID : String;   // Number received from MFC with the order to reject the package (ObjectID)
   END_VAR

   VAR
      s_FB_MFC_Sort_VIDResponse_ASCII { ExternalAccessible := 'False'; ExternalVisible := 'False'; ExternalWritable := 'False'; S7_SetPoint := 'False'} : "FB_MFC_Sort_VIDResponse_ASCII";   // VID message generator
      F_TRIG_PEC_EoS {InstructionName := 'F_TRIG'; LibVersion := '1.0'; ExternalAccessible := 'False'; ExternalVisible := 'False'; ExternalWritable := 'False'; S7_SetPoint := 'False'} : F_TRIG;   // Rising edge for photo eye
      sx_WaitForObjectID { ExternalAccessible := 'False'; ExternalVisible := 'False'; ExternalWritable := 'False'} : Bool;   // True - Parcel is in position, wait for information from MFC
      sx_WaitForDestination { ExternalAccessible := 'False'; ExternalVisible := 'False'; ExternalWritable := 'False'} : Bool;   // True - Parcel is in position, wait for information from MFC
      sx_WaitForParcel { ExternalAccessible := 'False'; ExternalVisible := 'False'; ExternalWritable := 'False'} : Bool;   // True - Information from MFC received , wait for parcel
      sx_ParcelReject { ExternalAccessible := 'False'; ExternalVisible := 'False'; ExternalWritable := 'False'} : Bool;   // True - The parcel is rejected by the MFC system
   END_VAR

   VAR_TEMP
      tudi_MFCRejectObjectID : UDInt;   // MFC Reject Object ID
   END_VAR


BEGIN
	(*
	----------------------------------------------------------------------------------------
	|                                                                                      |
	|  Copyright  2023             FORTNA Europe BV                                        |
	|  All Rights Reserved         Netherlands                                             |
	|                                                                                      |
	----------------------------------------------------------------------------------------
	Version history:
	Date        | Version   | Author       | Remark
	----------------------------------------------------------------------------------------
	28/06/2023  | 1.0       | S. Nikodem   | Release TIA 17 | DHL Munich 2023
	13/09/2023  | 1.1       | S. Nikodem   | Update interface
	13/03/2024  | 1.2       | S. Nieswiec  | Added to new baseline, block needs uptade after munich is finished
	*)

	REGION 1 - Triggers

	    // Rising edge - Parcel detected
	    #F_TRIG_PEC_EoS(CLK := #ix_PEC_EoS);

	END_REGION

	REGION 2 - Buttons

	    //Knee button
	    IF #ix_KneeButton AND #ix_PEC_EoS THEN

	        #sx_WaitForParcel := True;

	    END_IF;

	    //Reset button
	    //Reset after removing the package.
	    IF #ix_ResetButton AND #ix_PEC_EoS AND #sx_ParcelReject THEN
	        #sx_ParcelReject := False;
	    END_IF;

	END_REGION

	REGION 3 - Data

	    REGION 3.1 - Object ID

	        IF (#iqa_TrackingData[#i_UDT_PECUpdateConfiguration.Distance] > 0) THEN

	            //Match GIN with Object ID
	            IF NOT #ix_PEC_EoS                                                          // Parcel on the sensor
	                AND NOT "DB_GIN".GIN[#iqa_TrackingData[#i_UDT_PECUpdateConfiguration.Distance]].DHL.MFCMessage.Received.TemporaryParcelIdentifier  //The message for this GIN has not yet been received.
	                AND NOT (#iqs_MFCNewObjectID = '0')                                             // New Object ID
	            THEN

	                //Copy data from MFC
	                "DB_GIN".GIN[#iqa_TrackingData[#i_UDT_PECUpdateConfiguration.Distance]].DHL.ObjectID := #iqs_MFCNewObjectID;

	                //Temporary Parcel Identifier message with Object ID received
	                "DB_GIN".GIN[#iqa_TrackingData[#i_UDT_PECUpdateConfiguration.Distance]].DHL.MFCMessage.Received.TemporaryParcelIdentifier := True;
	                "DB_GIN".GIN[#iqa_TrackingData[#i_UDT_PECUpdateConfiguration.Distance]].General.Identification.GoodRead := True;

	                // Generate VID
	                #s_FB_MFC_Sort_VIDResponse_ASCII(is_ObjectID := #iqs_MFCNewObjectID,
	                                                 i_ActualTimeDTL := #idtl_ActualTime,
	                                                 iq_UDT_FifoHeader := #iq_UDT_FifoHeaderMFCMessage,
	                                                 iqs_FifoData := #iqs_FifoDataMFCMessage,
	                                                 iqdi_MessageSequenceNumber := #iqdi_MessageSequenceNumber);

	                //VID Response message generated
	                "DB_GIN".GIN[#iqa_TrackingData[#i_UDT_PECUpdateConfiguration.Distance]].DHL.MFCMessage.Sent.VIDResponse := True;

	                //Reset data in DB_MFC
	                #iqs_MFCNewObjectID := '0';

	                //Reset value
	                #sx_WaitForObjectID := False;

	            END_IF;

	        END_IF;


	    END_REGION

	    REGION 3.2 -Destination

	        IF (#iqa_TrackingData[#i_UDT_PECUpdateConfiguration.Distance] > 0) THEN

	            IF NOT #ix_PEC_EoS                                                              // Parcel on the sensor
	                AND NOT #sx_WaitForObjectID                                                 // Object ID received
	                AND "DB_GIN".GIN[#iqa_TrackingData[#i_UDT_PECUpdateConfiguration.Distance]].DHL.MFCMessage.Received.Destination                    //The message for this GIN has been received.
	            THEN

	                //Reset value
	                #sx_WaitForDestination := False;

	            END_IF;

	        END_IF;

	    END_REGION

	    REGION 3.3 - Parcel Reject

	        #tudi_MFCRejectObjectID := STRING_TO_UDINT(#is_MFCRejectObjectID);

	        IF (#iqa_TrackingData[#i_UDT_PECUpdateConfiguration.Distance] > 0) THEN

	            IF NOT #ix_PEC_EoS                                                          // Parcel on the sensor
	                AND NOT #sx_WaitForObjectID                                             // Object ID received
	                AND #tudi_MFCRejectObjectID > 0                       // New destination message from MFC reveived
	                AND ("DB_GIN".GIN[#iqa_TrackingData[#i_UDT_PECUpdateConfiguration.Distance]].DHL.ObjectID = #is_MFCRejectObjectID)
	                AND NOT "DB_GIN".GIN[#iqa_TrackingData[#i_UDT_PECUpdateConfiguration.Distance]].DHL.MFCMessage.Received.RejectParcel //The message for this GIN has not yet been received.
	            THEN

	                //Reject parcel received
	                "DB_GIN".GIN[#iqa_TrackingData[#i_UDT_PECUpdateConfiguration.Distance]].DHL.MFCMessage.Received.RejectParcel := True;

	                //Reset data in DB_MFC
	                #is_MFCRejectObjectID := '0';

	                //Reset value
	                #sx_WaitForDestination := False;

	                //Set value
	                #sx_ParcelReject := True;

	            END_IF;

	        END_IF;

	    END_REGION

	    //Hold conveyor if parcel is detected
	    IF #F_TRIG_PEC_EoS.Q THEN
	        #sx_WaitForObjectID := True;
	        #sx_WaitForDestination := True;
	        #sx_WaitForParcel := FALSE;
	    END_IF;

	    //Data received wait for parcel
	    IF NOT (#iqs_MFCNewObjectID = '0') THEN
	        #sx_WaitForParcel := True;
	    END_IF;

	    //Hold
	    #qx_ConveyorHold := NOT #sx_WaitForParcel AND (#sx_WaitForDestination OR #sx_ParcelReject);

	END_REGION

	REGION 4 - Lamp handling

	    //White lamp
	    //1 hz - Parcel on the sensor, waiting for data from MFC
	    //On - Waiting for a package
	    #qx_WhiteLamp := NOT #sx_ParcelReject AND (NOT #ix_PEC_EoS OR (#sx_WaitForObjectID AND "DB_Memory".Clock_1Hz));

	    //Blue lamp
	    //1 hz - Parcel reject
	    #qx_BlueLamp := #sx_ParcelReject AND "DB_Memory".Clock_1Hz;

	END_REGION
END_FUNCTION_BLOCK

FUNCTION_BLOCK "FB_EuchnerLockV2"
{ S7_Optimized_Access := 'TRUE' }
VERSION : 0.1
// ATTRIBUTES
// AUTO_NUMBER = True
// BLOCK_NUMBER = 96
// END_ATTRIBUTES
   VAR_INPUT
      ix_ButtonReset { ExternalAccessible := 'False'; ExternalVisible := 'False'; ExternalWritable := 'False'} : Bool;   // Reset button
      ix_ButtonRequest { ExternalAccessible := 'False'; ExternalVisible := 'False'; ExternalWritable := 'False'} : Bool;   // Request open button
      ix_IdCardAccessGranted { ExternalAccessible := 'False'; ExternalVisible := 'False'; ExternalWritable := 'False'} : Bool;   // Feedback from DHL- ID card ok - access granted
      ix_DoorClosed { ExternalAccessible := 'False'; ExternalVisible := 'False'; ExternalWritable := 'False'} : Bool;   // Feedback from lock - door is closed
      ix_BoltTongueClosed { ExternalAccessible := 'False'; ExternalVisible := 'False'; ExternalWritable := 'False'} : Bool;   // Feedback from lock - bolt tongue closed
      ix_SafelyLoced { ExternalAccessible := 'False'; ExternalVisible := 'False'; ExternalWritable := 'False'} : Bool;   // Feedback from lock - Safely locked
      ix_InternalErrorReset { ExternalAccessible := 'False'; ExternalVisible := 'False'; ExternalWritable := 'False'} : Bool;   // Internal error reset command from system control
      ix_LockFault { ExternalAccessible := 'False'; ExternalVisible := 'False'; ExternalWritable := 'False'} : Bool;   // Lock has an internal fault
      ix_SystemStopped { ExternalAccessible := 'False'; ExternalVisible := 'False'; ExternalWritable := 'False'} : Bool;   // Feedback from system - System is stopped
      ix_SafetyLockOK { ExternalAccessible := 'False'; ExternalVisible := 'False'; ExternalWritable := 'False'} : Bool;   // Safety lock status OK
      ix_SafetyLockAckReq { ExternalAccessible := 'False'; ExternalVisible := 'False'; ExternalWritable := 'False'} : Bool;   // Safety lock need acknowledgement
      ii_NumberOfLEDs { ExternalAccessible := 'False'; ExternalVisible := 'False'; ExternalWritable := 'False'} : Int;   // Number of programmable LEDs on lock
   END_VAR

   VAR_OUTPUT
      qx_StopSystem { ExternalAccessible := 'False'; ExternalVisible := 'False'; ExternalWritable := 'False'} : Bool;   // Signal to stop the system
      qx_ResetButtonLed { ExternalAccessible := 'False'; ExternalVisible := 'False'; ExternalWritable := 'False'} : Bool;   // Reset button lamp
      qx_RequestButtonLed { ExternalAccessible := 'False'; ExternalVisible := 'False'; ExternalWritable := 'False'} : Bool;   // Request button lamp
      qx_FaultReset { ExternalAccessible := 'False'; ExternalVisible := 'False'; ExternalWritable := 'False'} : Bool;   // Reset internal lock fault
      qx_SafetyReset { ExternalAccessible := 'False'; ExternalVisible := 'False'; ExternalWritable := 'False'} : Bool;   // Safety reset command after authorization
      qx_ReleaseLock { ExternalAccessible := 'False'; ExternalVisible := 'False'; ExternalWritable := 'False'} : Bool;   // Signal to safety logic to release lock
      q_UDT_Status { ExternalAccessible := 'False'; ExternalVisible := 'False'; ExternalWritable := 'False'} : "UDT_EuchnerLockStatusV2";   // Status structure
   END_VAR

   VAR
      s_R_TRIG_RequestButton {InstructionName := 'R_TRIG'; LibVersion := '1.0'; ExternalAccessible := 'False'; ExternalVisible := 'False'; ExternalWritable := 'False'; S7_SetPoint := 'False'} : R_TRIG;   // Rising edge trigger from reqest button
      s_F_TRIG_BoltTongueClosed {InstructionName := 'F_TRIG'; LibVersion := '1.0'; ExternalAccessible := 'False'; ExternalVisible := 'False'; ExternalWritable := 'False'; S7_SetPoint := 'False'} : F_TRIG;   // Falling edge trigger from bolt tongue
      s_F_TRIG_ReleaseLock {InstructionName := 'F_TRIG'; LibVersion := '1.0'; ExternalAccessible := 'False'; ExternalVisible := 'False'; ExternalWritable := 'False'; S7_SetPoint := 'False'} : F_TRIG;   // Falling edge trigger from release lock
      s_FB_TimerOnOffDelay { ExternalAccessible := 'False'; ExternalVisible := 'False'; ExternalWritable := 'False'; S7_SetPoint := 'False'} : "FB_TimerOnOffDelay";   // Function block to generate on signal delay - emergency request button
      s_FB_TimerOnOffDelay_ResetDelay { ExternalAccessible := 'False'; ExternalVisible := 'False'; ExternalWritable := 'False'; S7_SetPoint := 'False'} : "FB_TimerOnOffDelay";
      sx_Request { ExternalAccessible := 'False'; ExternalVisible := 'False'; ExternalWritable := 'False'} : Bool;   // Request to open the door
      sx_ReqMissingAccessRights { ExternalAccessible := 'False'; ExternalVisible := 'False'; ExternalWritable := 'False'} : Bool;   // Button access request triggered without permission from DHL
      sx_ResetMissingAccessRights { ExternalAccessible := 'False'; ExternalVisible := 'False'; ExternalWritable := 'False'} : Bool;   // Button Reset triggered without permission from DHL
      sx_DoorOpenedWithoutReq { ExternalAccessible := 'False'; ExternalVisible := 'False'; ExternalWritable := 'False'} : Bool;   // Doors were opened without request and permission
   END_VAR

   VAR CONSTANT
      c_Time : UDInt := 10000;
   END_VAR


BEGIN

	(*
	----------------------------------------------------------------------------------------
	|                                                                                      |
	|  Copyright  2023             FORTNA Europe BV                                        |
	|  All Rights Reserved         Netherlands                                             |
	|                                                                                      |
	----------------------------------------------------------------------------------------

	Version history:
	Date        | Version   | Author       | Remark
	----------------------------------------------------------------------------------------
	11/03/2022  | 0.1       | S.Nikodem    | first release MHS TIA 15.1
	24/08/2022  | 0.2       | K. Pokorski  | Change to Lock with key switch and only one LED
	11/10/2023  | 0.3       | M.Diebel     | first release Fortna TIA 17
	30/01/2024  | 0.4       | A. Bunzel    | Add logic for ID cards from DHL
	13/03/2024  | 0.5       | S. Nieswiec  | Changed name to V2
	*)

	REGION 1 - Request open

	    //Button
	    //Rising edge trigger
	    #s_R_TRIG_RequestButton(CLK := #ix_ButtonRequest);

	    // Flip-flop
	    IF #s_R_TRIG_RequestButton.Q AND #ix_IdCardAccessGranted THEN

	        IF #sx_Request THEN
	            #sx_Request := FALSE;
	        ELSE
	            #sx_Request := TRUE;
	        END_IF;

	    END_IF;

	    // Reset Flip-Flop
	    IF NOT #ix_BoltTongueClosed THEN
	        #sx_Request := FALSE;
	    END_IF;

	    //Stop system
	    #qx_StopSystem := #sx_Request;

	    //If system is stopped and is safe then open lock
	    #qx_ReleaseLock := (#sx_Request AND #ix_SystemStopped);

	END_REGION

	REGION 2 - Lamp controlling


	    CASE #ii_NumberOfLEDs OF
	        1:
	            //2.5Hz blinking during fault
	            IF #ix_LockFault THEN
	                #qx_ResetButtonLed := "mx_Clock_2.5Hz";
	                //2.5Hz blinking when ACK required
	            ELSIF #ix_SafetyLockAckReq THEN
	                #qx_ResetButtonLed := "mx_Clock_2.5Hz";
	                //1.0Hz blinking during open request
	            ELSIF #sx_Request AND NOT #ix_SystemStopped THEN
	                #qx_ResetButtonLed := "mx_Clock_1Hz";
	                // Solid when system stopped after request
	            ELSIF #sx_Request THEN
	                #qx_ResetButtonLed := TRUE;
	                // Solid when doors open
	            ELSIF (NOT #ix_SafelyLoced AND NOT #ix_BoltTongueClosed) THEN
	                #qx_ResetButtonLed := TRUE;
	                // Turn off when gate closed and acknowledged
	            ELSE
	                #qx_ResetButtonLed := FALSE;
	            END_IF;

	        2:
	            // Reset button LED - Blue
	            // Lamp active - Reset access is granted and reset request is active
	            // Lamp flashing - Error doors where opened without request
	            IF #sx_DoorOpenedWithoutReq AND NOT #ix_BoltTongueClosed THEN
	                #qx_ResetButtonLed := "mx_Clock_0.625Hz";
	            ELSIF #ix_IdCardAccessGranted AND #ix_SafetyLockAckReq THEN
	                #qx_ResetButtonLed := TRUE;
	            ELSE
	                #qx_ResetButtonLed := FALSE;
	            END_IF;

	            // Request button LED - White
	            // Lamp active - System is stopped and safety
	            // Lamp flashing 0.62Hz - Error doors where opened without request
	            // Lamp flashing 1HZ - Request is active, system still not save.
	            // Lamp flashing 2.5Hz - Access rights are granted, and it is possible to make entry request.
	            IF #sx_DoorOpenedWithoutReq AND NOT #ix_BoltTongueClosed THEN
	                #qx_RequestButtonLed := "mx_Clock_0.625Hz";
	            ELSIF (#sx_Request AND #ix_SystemStopped) OR NOT #ix_SafetyLockOK THEN
	                #qx_RequestButtonLed := TRUE;
	            ELSIF #sx_Request THEN
	                #qx_RequestButtonLed := "mx_Clock_1Hz";
	            ELSIF #ix_IdCardAccessGranted THEN
	                #qx_RequestButtonLed := "mx_Clock_2.5Hz";
	            ELSE
	                #qx_RequestButtonLed := FALSE;
	            END_IF;
	    END_CASE;

	END_REGION

	REGION 3 - Fault

	    //Triggers
	    #s_F_TRIG_BoltTongueClosed(CLK := #ix_BoltTongueClosed);
	    #s_F_TRIG_ReleaseLock(CLK := #qx_ReleaseLock);

	    // Alarm from unauthorized open request
	    IF #ix_ButtonRequest AND NOT #ix_IdCardAccessGranted THEN

	        #sx_ReqMissingAccessRights := TRUE;

	    END_IF;

	    // Alarm when Doors are opened from inside (red door handle) without request
	    IF NOT #qx_ReleaseLock AND NOT #s_F_TRIG_ReleaseLock.Q AND #s_F_TRIG_BoltTongueClosed.Q THEN
	        #sx_DoorOpenedWithoutReq := TRUE;
	    END_IF;

	    // Alarm from unauthorized reset request
	    IF NOT #ix_IdCardAccessGranted AND #ix_ButtonReset THEN
	        #sx_ResetMissingAccessRights := TRUE;
	    END_IF;

	END_REGION

	REGION 4 - Falut reset

	    // reset alarm from unauthorized open request
	    IF #ix_InternalErrorReset AND #sx_ReqMissingAccessRights THEN
	        #sx_ReqMissingAccessRights := FALSE;
	    END_IF;

	    // reset alarm when Doors are opened from inside (red door handle) without request
	    IF #ix_InternalErrorReset AND #sx_DoorOpenedWithoutReq THEN
	        #sx_DoorOpenedWithoutReq := FALSE;
	    END_IF;

	    // reset alarm from unauthorized reset request
	    IF #ix_InternalErrorReset AND #sx_ResetMissingAccessRights THEN
	        #sx_ResetMissingAccessRights := FALSE;
	    END_IF;

	    // extended reset signal for door lock when error exist
	    #s_FB_TimerOnOffDelay_ResetDelay(iudi_OnDelayTime := 0,
	                                     iudi_OffDelayTime := 3500,
	                                     ix_SignalToDelay := (#ix_LockFault) AND (#ix_IdCardAccessGranted) AND (#ix_ButtonReset));


	    // Set reset signal
	    #qx_FaultReset := #s_FB_TimerOnOffDelay_ResetDelay.qx_DelayedSignal;

	END_REGION
	REGION 5 - Reset safety command
	    // Command for safety reset
	    #qx_SafetyReset := #ix_IdCardAccessGranted AND #ix_SafetyLockAckReq AND #ix_ButtonReset;

	END_REGION
	REGION 6 - Status

	    // Copy status
	    #q_UDT_Status.LockFault := #ix_LockFault;
	    #q_UDT_Status.DoorClosed := #ix_DoorClosed;
	    #q_UDT_Status.DoorOpened := NOT #ix_DoorClosed;
	    #q_UDT_Status.ReqMissingAccessRights := #sx_ReqMissingAccessRights;
	    #q_UDT_Status.DoorOpenedWithoutReq := #sx_DoorOpenedWithoutReq;
	    #q_UDT_Status.ResetMissingAccessRights := #sx_ResetMissingAccessRights;
	    #q_UDT_Status.BoltTongueClosed := #ix_BoltTongueClosed;
	    #q_UDT_Status.Safelylocked := #ix_SafelyLoced;
	    #q_UDT_Status.SafetyLockAckReq := #ix_SafetyLockAckReq;

	END_REGION

END_FUNCTION_BLOCK

FUNCTION_BLOCK "FB_EncoderValue"
{ S7_Optimized_Access := 'TRUE' }
VERSION : 0.1
// ATTRIBUTES
// AUTO_NUMBER = True
// BLOCK_NUMBER = 95
// END_ATTRIBUTES
   VAR_INPUT
      i_UDT_EncoderConfiguration { ExternalAccessible := 'False'; ExternalVisible := 'False'; ExternalWritable := 'False'} : "UDT_EncoderConfigurationV2";   // Encoder configuration structure
      id_EncoderValue { ExternalAccessible := 'False'; ExternalVisible := 'False'; ExternalWritable := 'False'} : DInt;   // Encoder value
      ix_EncoderDirection { ExternalAccessible := 'False'; ExternalVisible := 'False'; ExternalWritable := 'False'} : Bool;   // True if encoder rotates forward, False if encoder rotates reverse
      ix_ConveyorRunningFwd { ExternalAccessible := 'False'; ExternalVisible := 'False'; ExternalWritable := 'False'} : Bool;   // True when the conveyor is running in the forward direction
      ix_ConveyorRunningRvs { ExternalAccessible := 'False'; ExternalVisible := 'False'; ExternalWritable := 'False'} : Bool;   // True when the conveyor is running in the reverse direction
   END_VAR

   VAR_OUTPUT
      q_UDT_Status { ExternalAccessible := 'False'; ExternalVisible := 'False'; ExternalWritable := 'False'} : "UDT_EncoderStatusV2";   // Encoder status structure
      qi_ActualSpeed { ExternalAccessible := 'False'; ExternalVisible := 'False'; ExternalWritable := 'False'} : Int;   // Calculated speed [mm/sec]
      qi_Displacement { ExternalAccessible := 'False'; ExternalVisible := 'False'; ExternalWritable := 'False'} : Int;   // Calculated displacement [cm]
   END_VAR

   VAR_IN_OUT
      iq_UDT_EquipmentControl : "UDT_EquipmentControl";   // Equipment control structure
      iq_UDT_Statistics : "UDT_EncoderStatisticsV2";   // Statistics structure
   END_VAR

   VAR
      s_FB_SamplingTime { ExternalAccessible := 'False'; ExternalVisible := 'False'; ExternalWritable := 'False'; S7_SetPoint := 'False'} : "FB_TimerOnOffDelay";   // Error detection timer
      s_FB_RunningFeedbackError { ExternalAccessible := 'False'; ExternalVisible := 'False'; ExternalWritable := 'False'; S7_SetPoint := 'False'} : "FB_TimerOnOffDelay";   // Error detection timer
      R_TRIG_RunningFeedbackError {InstructionName := 'R_TRIG'; LibVersion := '1.0'; ExternalAccessible := 'False'; ExternalVisible := 'False'; ExternalWritable := 'False'; S7_SetPoint := 'False'} : R_TRIG;   // Rising edge trigger of running feedback error
      R_TRIG_InvalidValue {InstructionName := 'R_TRIG'; LibVersion := '1.0'; ExternalAccessible := 'False'; ExternalVisible := 'False'; ExternalWritable := 'False'; S7_SetPoint := 'False'} : R_TRIG;   // Rising edge trigger of invalid value
      R_TRIG_NoDirection {InstructionName := 'R_TRIG'; LibVersion := '1.0'; ExternalAccessible := 'False'; ExternalVisible := 'False'; ExternalWritable := 'False'; S7_SetPoint := 'False'} : R_TRIG;   // Rising edge trigger of no direction command
      s_UDT_Status { ExternalAccessible := 'False'; ExternalVisible := 'False'; ExternalWritable := 'False'; S7_SetPoint := 'False'} : "UDT_EncoderStatusV2";   // Encoder status structure
      sa_EncoderData { ExternalAccessible := 'False'; ExternalVisible := 'False'; ExternalWritable := 'False'} : Array[1..10] of DInt;   // Encoder data in array
      sa_SpeedData { ExternalAccessible := 'False'; ExternalVisible := 'False'; ExternalWritable := 'False'} : Array[1..20] of Struct   // Encoder sampled distance and time in array
         Distance { ExternalAccessible := 'False'; ExternalVisible := 'False'; ExternalWritable := 'False'} : Int;   // Distance [mm]
         "Time" { ExternalAccessible := 'False'; ExternalVisible := 'False'; ExternalWritable := 'False'} : UDInt;   // Time [sec]
      END_STRUCT;
      slr_FormDisplacement { ExternalAccessible := 'False'; ExternalVisible := 'False'; ExternalWritable := 'False'} : LReal;   // Conveyor displacement [cm]
      slr_Correction { ExternalAccessible := 'False'; ExternalVisible := 'False'; ExternalWritable := 'False'} : LReal;   // Correction [cm]
      sdi_Value { ExternalAccessible := 'False'; ExternalVisible := 'False'; ExternalWritable := 'False'} : DInt;   // Value from encoder card
      sdi_OldValue { ExternalAccessible := 'False'; ExternalVisible := 'False'; ExternalWritable := 'False'} : DInt;   // Old value from encoder card
      sdi_Delta { ExternalAccessible := 'False'; ExternalVisible := 'False'; ExternalWritable := 'False'} : DInt;   // Encoder value per cycle
      si_StatusMoveBLKVariant { ExternalAccessible := 'False'; ExternalVisible := 'False'; ExternalWritable := 'False'} : Int;   // Move BLK status
      si_SampleDisplacement { ExternalAccessible := 'False'; ExternalVisible := 'False'; ExternalWritable := 'False'} : Int;   // Travel the distance for one sample
      si_ActualSpeed { ExternalAccessible := 'False'; ExternalVisible := 'False'; ExternalWritable := 'False'} : Int;   // Actual speed [mm/sec]
      sx_InvalidValue { ExternalAccessible := 'False'; ExternalVisible := 'False'; ExternalWritable := 'False'} : Bool;   // Invalid encoder value
   END_VAR

   VAR_TEMP
      ti_TotalTime : UDInt;   // Total sampled time
      ti_TotalDistance : DInt;   // Total sampled distance
      ti_Displacement : Int;   // Conveyor displacement [cm]
      ti_ArraySize : Int;   // Array size
      ti_LoopActulaSpeed : Int;   // Loop counter
   END_VAR


BEGIN
	(*
	----------------------------------------------------------------------------------------
	|                                                                                      |
	|  Copyright  2023             FORTNA Europe BV                                        |
	|  All Rights Reserved         Netherlands                                             |
	|                                                                                      |
	----------------------------------------------------------------------------------------

	Version history:
	Date        | Version   | Author       | Remark
	----------------------------------------------------------------------------------------
	29/03/2023  | 1.0       | S. Nikodem   | Release TIA 17 | DHL Munich 2023
	12/03/2024  | 1.1       | S. Nieswiec  | Updated for new baseline
	*)

	REGION 1 - Triggers

	    //Conveyor is not running
	    #R_TRIG_NoDirection(CLK := NOT #ix_ConveyorRunningFwd AND NOT #ix_ConveyorRunningRvs);

	    //Invalid value error
	    #R_TRIG_InvalidValue(CLK := #s_UDT_Status.InvalidValue);

	END_REGION

	REGION 1 - Displacement

	    //Check if encoder value is in range
	    IF #id_EncoderValue > #i_UDT_EncoderConfiguration.EncoderMaxValue THEN

	        //Set fault
	        #sx_InvalidValue := TRUE;

	    ELSE

	        //Copy encoder value
	        #sdi_Value := #id_EncoderValue;

	        //Reset fault
	        #sx_InvalidValue := FALSE;

	    END_IF;

	    REGION 1.1 - Encoder data

	        IF (#sdi_OldValue <> #sdi_Value)
	            AND NOT #s_UDT_Status.InvalidValue
	        THEN

	            //Check array size
	            #ti_ArraySize := "FC_GetNrOfArrayEl"(iv_Array := #sa_EncoderData);

	            // Switch data in the array
	            #si_StatusMoveBLKVariant := MOVE_BLK_VARIANT(SRC := #sa_EncoderData, COUNT := INT_TO_UINT(#ti_ArraySize - 1), SRC_INDEX := 0, DEST_INDEX := 1, DEST => #sa_EncoderData);

	            //Save data in array
	            #sa_EncoderData[1] := #sdi_Value;

	            //Conveyor is running in the forward direction
	            IF #ix_EncoderDirection THEN

	                IF #sa_EncoderData[1] < #sa_EncoderData[2] THEN

	                    //Rollover
	                    #sdi_Delta := #i_UDT_EncoderConfiguration.EncoderMaxValue - #sa_EncoderData[2] + #sa_EncoderData[1];

	                ELSE

	                    #sdi_Delta := #sa_EncoderData[1] - #sa_EncoderData[2];

	                END_IF;

	            END_IF;

	            //Conveyor is running in the reverse direction
	            IF #ix_EncoderDirection THEN

	                IF #sa_EncoderData[1] > #sa_EncoderData[2] THEN

	                    //Rollover
	                    #sdi_Delta := #i_UDT_EncoderConfiguration.EncoderMaxValue - #sa_EncoderData[1] + #sa_EncoderData[2];

	                ELSE

	                    #sdi_Delta := #sa_EncoderData[2] - #sa_EncoderData[1];

	                END_IF;

	            END_IF;

	        END_IF;

	    END_REGION

	    REGION 1.2 - mm per encoder incremental

	        //Count up value in mm ,
	        // Displacement is calculated using actual conveyor speed and the previous PLC cycle scan time
	        #slr_FormDisplacement := DINT_TO_LREAL(#sdi_Delta) * #i_UDT_EncoderConfiguration.mmPerIncrement / 10.0;

	        //Accumulate the rest of the calculated value
	        #slr_Correction := FRAC(#slr_FormDisplacement) + #slr_Correction;

	        // The actual displacement is a sum of complete parts of the displacement and correction variables
	        #ti_Displacement := DINT_TO_INT(TRUNC(#slr_FormDisplacement) + TRUNC(#slr_Correction));

	        // Correction incrementation or decremantation if it exceeds 1 or -1 in case of negative speed
	        IF (#slr_Correction >= 1)
	        THEN

	            #slr_Correction -= 1;

	        ELSIF (#slr_Correction <= -1)
	        THEN

	            #slr_Correction += 1;

	        END_IF;

	        //Reset delta value
	        #sdi_Delta := 0;

	    END_REGION

	END_REGION

	REGION 2- Actual speed

	    //Check array size
	    #ti_ArraySize := "FC_GetNrOfArrayEl"(iv_Array := #sa_SpeedData);

	    //Sampling time
	    #s_FB_SamplingTime(iudi_OnDelayTime := #i_UDT_EncoderConfiguration.SamplingTime,
	                       ix_SignalToDelay := (#ix_ConveyorRunningFwd OR #ix_ConveyorRunningRvs) AND NOT #s_FB_SamplingTime.qx_DelayedSignal);

	    //Save displacemnt only when conveyor is running
	    IF #ix_ConveyorRunningFwd OR #ix_ConveyorRunningRvs THEN
	        #si_SampleDisplacement += #ti_Displacement;
	    END_IF;

	    //Saving data every sampling time
	    IF #s_FB_SamplingTime.qx_DelayedSignal THEN

	        // Switch data in the array
	        #si_StatusMoveBLKVariant := MOVE_BLK_VARIANT(SRC := #sa_SpeedData, COUNT := INT_TO_UINT(#ti_ArraySize - 1), SRC_INDEX := 0, DEST_INDEX := 1, DEST => #sa_SpeedData);

	        //Copy data to array
	        //Save distance value in mm
	        #sa_SpeedData[1].Distance := #si_SampleDisplacement;
	        //Save time value in ms
	        #sa_SpeedData[1]."Time" := (LREAL_TO_UDINT(#s_FB_SamplingTime.qlr_ActualTime));

	        //Reset varaible
	        #si_SampleDisplacement := 0;

	    END_IF;

	    //Calculate the speed according to the data in the array
	    FOR #ti_LoopActulaSpeed := 1 TO #ti_ArraySize DO

	        //[mm]
	        #ti_TotalDistance += ABS(#sa_SpeedData[#ti_LoopActulaSpeed].Distance);
	        //[sec]
	        #ti_TotalTime += #sa_SpeedData[#ti_LoopActulaSpeed]."Time";

	        //Reset data in array
	        IF #R_TRIG_NoDirection.Q THEN

	            #sa_SpeedData[#ti_LoopActulaSpeed].Distance := 0;
	            #sa_SpeedData[#ti_LoopActulaSpeed]."Time" := 0;

	        END_IF;

	    END_FOR;

	    //Actual speed in mm/sec
	    #si_ActualSpeed := DINT_TO_INT((#ti_TotalDistance / (UDINT_TO_DINT(#ti_TotalTime) / 1000)));

	END_REGION

	REGION 3 - Error

	    REGION 3.1 - Running feedback error

	        //Timer
	        #s_FB_RunningFeedbackError(iudi_OnDelayTime := #i_UDT_EncoderConfiguration.ErrorFilter,
	                                   ix_SignalToDelay := (#ix_ConveyorRunningFwd OR #ix_ConveyorRunningRvs) AND (#sdi_OldValue = #sdi_Value));

	        //Save last encoder value
	        #sdi_OldValue := #sdi_Value;

	        //Trigger from error signal
	        #R_TRIG_RunningFeedbackError(CLK := #s_FB_RunningFeedbackError.qx_DelayedSignal);

	        //Set running feedback error
	        IF #R_TRIG_RunningFeedbackError.Q THEN
	            #s_UDT_Status.RunningFeedbackError := True;
	        END_IF;

	    END_REGION

	    REGION 3.2 - Invalid Value error

	        //Set invalid value error
	        IF #sx_InvalidValue THEN
	            #s_UDT_Status.InvalidValue := True;
	        END_IF;

	    END_REGION

	    REGION 3.3 - Reset

	        //Reset error
	        IF #iq_UDT_EquipmentControl.Command.Reset THEN
	            #s_UDT_Status.RunningFeedbackError := False;
	            #s_UDT_Status.InvalidValue := False;
	        END_IF;

	    END_REGION

	END_REGION

	REGION 4 - Statistics

	    // Running feedback error statistics
	    IF #s_UDT_Status.RunningFeedbackError
	        OR #iq_UDT_EquipmentControl.Command.ResetData                                         // Reset statistics
	    THEN

	        "FC_Statistics"(ix_Reset := #iq_UDT_EquipmentControl.Command.ResetData,               // Reset statistics input
	                        ix_Activate := #s_UDT_Status.RunningFeedbackError,                    // Activate statistics functions input
	                        ix_RTrigActivate := #R_TRIG_RunningFeedbackError.Q,                   // Statistics active trigger
	                        iqUDT_Statistics := #iq_UDT_Statistics.RunningFeedbackError);        // Statistics values output

	    END_IF;

	    // Invalid Value statistics
	    IF #s_UDT_Status.InvalidValue
	        OR #iq_UDT_EquipmentControl.Command.ResetData                                         // Reset statistics
	    THEN

	        "FC_Statistics"(ix_Reset := #iq_UDT_EquipmentControl.Command.ResetData,               // Reset statistics input
	                        ix_Activate := #s_UDT_Status.InvalidValue,                            // Activate statistics functions input
	                        ix_RTrigActivate := #R_TRIG_InvalidValue.Q,                           // Statistics active trigger
	                        iqUDT_Statistics := #iq_UDT_Statistics.InvalidValue);                // Statistics values output

	    END_IF;

	END_REGION

	REGION 5 - Outputs

	    //Check motor direction
	    IF #ix_ConveyorRunningFwd THEN

	        //Actual speed
	        #qi_ActualSpeed := #si_ActualSpeed;
	        //Displacement
	        #qi_Displacement := #ti_Displacement;

	    ELSIF #ix_ConveyorRunningRvs THEN

	        //Actual speed
	        #qi_ActualSpeed := #si_ActualSpeed * -1;
	        //Displacement
	        #qi_Displacement := #ti_Displacement * -1;

	    ELSE

	        //Actual speed
	        #qi_ActualSpeed := 0;
	        //Displacement
	        #qi_Displacement := 0;

	    END_IF;

	    //Copy value to output
	    //Status
	    #q_UDT_Status := #s_UDT_Status;


	END_REGION

END_FUNCTION_BLOCK

FUNCTION_BLOCK "FB_ABSwitch"
{ S7_Optimized_Access := 'TRUE' }
VERSION : 0.1
// ATTRIBUTES
// AUTO_NUMBER = True
// BLOCK_NUMBER = 87
// END_ATTRIBUTES
   VAR_INPUT
      iUDT_ABSwitchConfig { ExternalAccessible := 'False'; ExternalVisible := 'False'; ExternalWritable := 'False'} : "UDT_ABSwitchConfiguration";   // AB Switch Configuration structure
      ix_SafetyOk { ExternalAccessible := 'False'; ExternalVisible := 'False'; ExternalWritable := 'False'} : Bool;   // TRUE when Safety Circuit of the Conveyor is healthy
      ix_PRXUp { ExternalAccessible := 'False'; ExternalVisible := 'False'; ExternalWritable := 'False'} : Bool;   // TRUE when upper position sensor is not covered
      ix_PRXDown { ExternalAccessible := 'False'; ExternalVisible := 'False'; ExternalWritable := 'False'} : Bool;   // TRUE when lower position sensor is not covered
      ix_PRXBrkUp { ExternalAccessible := 'False'; ExternalVisible := 'False'; ExternalWritable := 'False'} : Bool;   // TRUE when sensor to slow down the speed is not covered
      ix_PRXBrkDwn { ExternalAccessible := 'False'; ExternalVisible := 'False'; ExternalWritable := 'False'} : Bool;   // TRUE when sensor to slow down the speed is not covered
      ix_LSUp { ExternalAccessible := 'False'; ExternalVisible := 'False'; ExternalWritable := 'False'} : Bool;   // TRUE when upper limit sensor is not covered
      ix_LSDwn { ExternalAccessible := 'False'; ExternalVisible := 'False'; ExternalWritable := 'False'} : Bool;   // TRUE when lower limit sensor is not covered
      ix_PECFreUp { ExternalAccessible := 'False'; ExternalVisible := 'False'; ExternalWritable := 'False'} : Bool;   // TRUE when nothing is within the range of the motion sensor
      ix_PECFreDwn { ExternalAccessible := 'False'; ExternalVisible := 'False'; ExternalWritable := 'False'} : Bool;   // TRUE when nothing is within the range of the motion sensor
      ix_SSMan { ExternalAccessible := 'False'; ExternalVisible := 'False'; ExternalWritable := 'False'} : Bool;   // TRUE when on Local Controll Panel switch [1] Manual; [0] Automatic
      ix_PBDwn { ExternalAccessible := 'False'; ExternalVisible := 'False'; ExternalWritable := 'False'} : Bool;   // TRUE when Local Control Panel switch Down is on
      ix_PBUp { ExternalAccessible := 'False'; ExternalVisible := 'False'; ExternalWritable := 'False'} : Bool;   // TRUE when Local Control Panel switch Up is on
      ix_PBRst { ExternalAccessible := 'False'; ExternalVisible := 'False'; ExternalWritable := 'False'} : Bool;   // TRUE when Local Control Panel reset is on
      ix_HardwareOk { ExternalAccessible := 'False'; ExternalVisible := 'False'; ExternalWritable := 'False'} : Bool;   // TRUE when hardware is Ok
      ii_Mode { ExternalAccessible := 'False'; ExternalVisible := 'False'; ExternalWritable := 'False'} : Int;   // Mode - [1] Upper position [2] Lower position
      ix_ChangeModeSignal { ExternalAccessible := 'False'; ExternalVisible := 'False'; ExternalWritable := 'False'} : Bool;   // TRUE when change mode command active
   END_VAR

   VAR_OUTPUT
      qUDT_HMIStatus { ExternalAccessible := 'False'; ExternalVisible := 'False'; ExternalWritable := 'False'} : "UDT_ABSwitchStatus";   // HMI status structure
      qUDT_Status { ExternalAccessible := 'False'; ExternalVisible := 'False'; ExternalWritable := 'False'} : "UDT_CommonStatus";   // Common status structure
      qx_ExternalHold { ExternalAccessible := 'False'; ExternalVisible := 'False'; ExternalWritable := 'False'} : Bool;   // External hold for AB Switch belt
   END_VAR

   VAR_IN_OUT
      iqUDT_EquipmentControl : "UDT_EquipmentControl";   // Equipment control structure
      iqUDT_ABSwitchInterface : "UDT_ConveyorInterface";   // Interface AB Switch motor
      iqUDT_Statistics : "UDT_ABSwitchStatistics";   // Statistics structure
   END_VAR

   VAR
      sUDT_HMIStatus { ExternalAccessible := 'False'; ExternalVisible := 'False'; ExternalWritable := 'False'; S7_SetPoint := 'False'} : "UDT_ABSwitchStatus";   // HMI status structure
      sUDT_StatusOld { ExternalAccessible := 'False'; ExternalVisible := 'False'; ExternalWritable := 'False'; S7_SetPoint := 'False'} : "UDT_CommonStatus";   // Common status structure
      sUDT_Status { ExternalAccessible := 'False'; ExternalVisible := 'False'; ExternalWritable := 'False'; S7_SetPoint := 'False'} : "UDT_CommonStatus";   // Common status structure
      Jog_Enable { ExternalAccessible := 'False'; ExternalVisible := 'False'; ExternalWritable := 'False'; S7_SetPoint := 'False'} : "FB_TimerOnOffDelay";   // Filtering lower jam photo eye signal
      SwitchingTime { ExternalAccessible := 'False'; ExternalVisible := 'False'; ExternalWritable := 'False'; S7_SetPoint := 'False'} : "FB_TimerOnOffDelay";   // Switching time
      R_TRIG_ManualMode {InstructionName := 'R_TRIG'; LibVersion := '1.0'; ExternalAccessible := 'False'; ExternalVisible := 'False'; ExternalWritable := 'False'; S7_SetPoint := 'False'} : R_TRIG;   // Rising edge trigger manual mode
      R_TRIG_ManualJogUp {InstructionName := 'R_TRIG'; LibVersion := '1.0'; ExternalAccessible := 'False'; ExternalVisible := 'False'; ExternalWritable := 'False'; S7_SetPoint := 'False'} : R_TRIG;   // Rising edge trigger manual jog mode command
      R_TRIG_ManualJogDown {InstructionName := 'R_TRIG'; LibVersion := '1.0'; ExternalAccessible := 'False'; ExternalVisible := 'False'; ExternalWritable := 'False'; S7_SetPoint := 'False'} : R_TRIG;   // Rising edge trigger manual jog mode command
      R_TRIG_DownTime {InstructionName := 'R_TRIG'; LibVersion := '1.0'; ExternalAccessible := 'False'; ExternalVisible := 'False'; ExternalWritable := 'False'; S7_SetPoint := 'False'} : R_TRIG;   // Rising edge trigger VSU is stopped
      R_TRIG_Error {InstructionName := 'R_TRIG'; LibVersion := '1.0'; ExternalAccessible := 'False'; ExternalVisible := 'False'; ExternalWritable := 'False'; S7_SetPoint := 'False'} : R_TRIG;   // Rising edge trigger for Error
      R_TRIG_UPSwA_Error {InstructionName := 'R_TRIG'; LibVersion := '1.0'; ExternalAccessible := 'False'; ExternalVisible := 'False'; ExternalWritable := 'False'; S7_SetPoint := 'False'} : R_TRIG;   // Rising edge trigger for Upper switch area error
      R_TRIG_LowSwA_Error {InstructionName := 'R_TRIG'; LibVersion := '1.0'; ExternalAccessible := 'False'; ExternalVisible := 'False'; ExternalWritable := 'False'; S7_SetPoint := 'False'} : R_TRIG;   // Rising edge trigger for Lower switch area error
      R_TRIG_UpTime {InstructionName := 'R_TRIG'; LibVersion := '1.0'; ExternalAccessible := 'False'; ExternalVisible := 'False'; ExternalWritable := 'False'; S7_SetPoint := 'False'} : R_TRIG;   // Rising edge trigger AB switch is running automatic
      R_TRIG_RestartFromError {InstructionName := 'R_TRIG'; LibVersion := '1.0'; ExternalAccessible := 'False'; ExternalVisible := 'False'; ExternalWritable := 'False'; S7_SetPoint := 'False'} : R_TRIG;   // Rising edge trigger Restart from error
      F_TRIG_PECBrakeUp {InstructionName := 'F_TRIG'; LibVersion := '1.0'; ExternalAccessible := 'False'; ExternalVisible := 'False'; ExternalWritable := 'False'; S7_SetPoint := 'False'} : F_TRIG;   // Falling edge trigger for PEC brake up
      F_TRIG_PECBrakeDown {InstructionName := 'F_TRIG'; LibVersion := '1.0'; ExternalAccessible := 'False'; ExternalVisible := 'False'; ExternalWritable := 'False'; S7_SetPoint := 'False'} : F_TRIG;   // Falling edge trigger for PEC brake down
      F_TRIG_PECUp {InstructionName := 'F_TRIG'; LibVersion := '1.0'; ExternalAccessible := 'False'; ExternalVisible := 'False'; ExternalWritable := 'False'; S7_SetPoint := 'False'} : F_TRIG;   // Falling edge trigger for PEC up position
      F_TRIG_PECDown {InstructionName := 'F_TRIG'; LibVersion := '1.0'; ExternalAccessible := 'False'; ExternalVisible := 'False'; ExternalWritable := 'False'; S7_SetPoint := 'False'} : F_TRIG;   // Falling edge trigger for PEC down position
      R_TRIG_PreStartSemiAutomaticUp {InstructionName := 'F_TRIG'; LibVersion := '1.0'; ExternalAccessible := 'False'; ExternalVisible := 'False'; ExternalWritable := 'False'; S7_SetPoint := 'False'} : F_TRIG;   // Falling edge trigger for Pre start semi automatic up signal
      R_TRIG_PreStartSemiAutomaticDown {InstructionName := 'F_TRIG'; LibVersion := '1.0'; ExternalAccessible := 'False'; ExternalVisible := 'False'; ExternalWritable := 'False'; S7_SetPoint := 'False'} : F_TRIG;   // Falling edge trigger for Pre start semi automatic down signal
      ss_ABSwitch_Interface { ExternalAccessible := 'False'; ExternalVisible := 'False'; ExternalWritable := 'False'} : Struct   // VSU interface static structure
         Positioning { ExternalAccessible := 'False'; ExternalVisible := 'False'; ExternalWritable := 'False'} : Bool;
         SemiAutomatic { ExternalAccessible := 'False'; ExternalVisible := 'False'; ExternalWritable := 'False'} : Bool;
         Manual { ExternalAccessible := 'False'; ExternalVisible := 'False'; ExternalWritable := 'False'} : Bool;
         RunEnabled { ExternalAccessible := 'False'; ExternalVisible := 'False'; ExternalWritable := 'False'} : Bool;
      END_STRUCT;
      sx_StartReceived { ExternalAccessible := 'False'; ExternalVisible := 'False'; ExternalWritable := 'False'} : Bool;   // Start command received from system
      sx_Ready { ExternalAccessible := 'False'; ExternalVisible := 'False'; ExternalWritable := 'False'} : Bool;   // Conveyor Ready to operate in Automatic mode
      sx_SemiAutomatic { ExternalAccessible := 'False'; ExternalVisible := 'False'; ExternalWritable := 'False'} : Bool;   // Running in semi automatic
      sx_PreStartManual { ExternalAccessible := 'False'; ExternalVisible := 'False'; ExternalWritable := 'False'} : Bool;   // Pre conditions to run conveyor in manual mode
      sx_Stopping { ExternalAccessible := 'False'; ExternalVisible := 'False'; ExternalWritable := 'False'} : Bool;   // Stopping is active, first reach position
      sx_SwitchEnable { ExternalAccessible := 'False'; ExternalVisible := 'False'; ExternalWritable := 'False'} : Bool;   // Switching conditions
      sx_UpRequest { ExternalAccessible := 'False'; ExternalVisible := 'False'; ExternalWritable := 'False'} : Bool;   // Request upper outfeed position for actual parcel
      sx_DownRequest { ExternalAccessible := 'False'; ExternalVisible := 'False'; ExternalWritable := 'False'} : Bool;   // Request lower outfeed position for actual parcel
      sx_ActualPositionUP { ExternalAccessible := 'False'; ExternalVisible := 'False'; ExternalWritable := 'False'} : Bool;   // Actual position is up
      sx_ActualPositionDown { ExternalAccessible := 'False'; ExternalVisible := 'False'; ExternalWritable := 'False'} : Bool;   // Actual position is down
      sx_CombinedJogUp { ExternalAccessible := 'False'; ExternalVisible := 'False'; ExternalWritable := 'False'} : Bool;   // Combined signal of jogging buttons
      sx_CombinedJogDown { ExternalAccessible := 'False'; ExternalVisible := 'False'; ExternalWritable := 'False'} : Bool;   // Combined signal of jogging buttons
      sx_RestartFromError { ExternalAccessible := 'False'; ExternalVisible := 'False'; ExternalWritable := 'False'} : Bool;   // After an error has occurred the action to be done before resuming normal operation
      sx_Jog { ExternalAccessible := 'False'; ExternalVisible := 'False'; ExternalWritable := 'False'} : Bool;   // Off delayed signal Jogging was activated
      sx_ConfigurationError { ExternalAccessible := 'False'; ExternalVisible := 'False'; ExternalWritable := 'False'} : Bool;   // Commissioning: configuration of parameters is wrong
      sx_JogUp { ExternalAccessible := 'False'; ExternalVisible := 'False'; ExternalWritable := 'False'} : Bool;   // AB Switch in manual mode - jog up
      sx_JogDown { ExternalAccessible := 'False'; ExternalVisible := 'False'; ExternalWritable := 'False'} : Bool;   // AB Switch in manual mode - jog down
      sx_ABSwitchSlowSpeedUp { ExternalAccessible := 'False'; ExternalVisible := 'False'; ExternalWritable := 'False'} : Bool;   // Slow down the speed when AB Switch is going up
      sx_ABSwitchSlowSpeedDown { ExternalAccessible := 'False'; ExternalVisible := 'False'; ExternalWritable := 'False'} : Bool;   // Slow down the speed when AB Switch is going down
      sx_UpperPositionReached { ExternalAccessible := 'False'; ExternalVisible := 'False'; ExternalWritable := 'False'} : Bool;   // AB Switch is in upper position
      sx_LowerPositionReached { ExternalAccessible := 'False'; ExternalVisible := 'False'; ExternalWritable := 'False'} : Bool;   // AB Switch is in lower position
      sx_PreStartSemiAutomaticUp { ExternalAccessible := 'False'; ExternalVisible := 'False'; ExternalWritable := 'False'} : Bool;   // Pre conditions to run conveyor in semi automatic up mode
      sx_PreStartSemiAutomaticDown { ExternalAccessible := 'False'; ExternalVisible := 'False'; ExternalWritable := 'False'} : Bool;   // Pre conditions to run conveyor in semi automatic down  mode
   END_VAR

   VAR_TEMP
      ti_ActiveSensor : Int;   // Active sensor counter
   END_VAR

   VAR CONSTANT
      ci_UpperPosition : Int := 1;   // Upper position number
      ci_LowerPosition : Int := 2;   // Lower position number
   END_VAR


BEGIN
	(*
	----------------------------------------------------------------------------------------
	|                                                                                      |
	|  Copyright  2023             FORTNA Europe BV                                        |
	|  All Rights Reserved         Netherlands                                             |
	|                                                                                      |
	----------------------------------------------------------------------------------------
	Version history:
	Date        | Version   | Author       | Remark
	----------------------------------------------------------------------------------------
	19/05/2023  | 1.0       | S. Nikodem   | Release TIA 17 | DHL Munich 2023
	19/12/2023  | 1.1       | S. Nikodem   | On site update
	09/02/2024  | 1.2       | P.Gryszczyk  | Gap Down sensor invert
	02/03/2024  | 1.3       | P.Gryszczyk  | HMI Lower Upper Position invert
	12/03/2024  | 1.4       | S. Nieswiec  | Addjusting to naming standard
	*)

	REGION 1 - Initial

	    REGION 1.1 - Triggers

	        // Detecting rising edge on manual mode Or from Equipment Control
	        #R_TRIG_ManualMode(CLK := #sUDT_Status.Manual);

	        // Rising edge trigger running
	        #R_TRIG_UpTime(CLK := #sx_SemiAutomatic AND #sx_Ready);

	        // Detecting rising edge AB switch stopped
	        #R_TRIG_DownTime(CLK := #sx_SemiAutomatic AND NOT #sx_Ready);

	        // Detecting rising edge on AB switch error
	        #R_TRIG_Error(CLK := #sUDT_Status.Error);

	        // Detecting rising edge on start of the restart from error sequence
	        #R_TRIG_RestartFromError(CLK := #sx_RestartFromError);

	    END_REGION

	    REGION 1.2 - Filters

	        // Time to start without start warning while jogging
	        #Jog_Enable(iudi_OffDelayTime := #iUDT_ABSwitchConfig.JogNoHornTime,
	                    ix_SignalToDelay := #sx_Jog);

	    END_REGION

	    REGION 1.3 - Switching conditions

	        #sx_SwitchEnable := NOT #iqUDT_ABSwitchInterface.VFDRunning;

	    END_REGION

	    REGION 1.4 - Positioning

	        // To add manual mode

	        #ss_ABSwitch_Interface.Positioning := #iqUDT_ABSwitchInterface.ActualSpeed <> 0
	        AND #sx_SemiAutomatic
	        AND NOT #iqUDT_ABSwitchInterface.InternalErrorVFD;

	    END_REGION

	    REGION 1.5 - Position

	        #sx_ActualPositionUP := NOT #ss_ABSwitch_Interface.Positioning                              // The positioning is not active
	        AND NOT #ix_PRXUp;                                                          // And the position sensor signals

	        #sx_ActualPositionDown := NOT #ss_ABSwitch_Interface.Positioning                            // The positioning is not active
	        AND NOT #ix_PRXDown;                                                        // And the position sensor signals

	    END_REGION

	END_REGION

	REGION 2 - Errors

	    REGION 2.1 - Reset errors

	        //Global reset
	        IF #iqUDT_EquipmentControl.Command.Reset                                       // Reset
	        THEN
	            // Switch area
	            IF #sUDT_HMIStatus.Specific.UpperSwitchAreaError                            // Upper jam error is active
	                AND #ix_PECFreUp                                                       // Upper jam sensor is free
	            THEN

	                #sUDT_HMIStatus.Specific.UpperSwitchAreaError := FALSE;                 // reset error

	            END_IF;

	            IF #sUDT_HMIStatus.Specific.LowerSwitchAreaError                            // lower jam error is active
	                AND #ix_PECFreDwn                                                     // Lower jam sensor is free
	            THEN

	                #sUDT_HMIStatus.Specific.LowerSwitchAreaError := FALSE;                 // reset error

	            END_IF;

	        END_IF;

	        //Local reset
	        IF #ix_PBRst THEN

	            // Switch area
	            IF #sUDT_HMIStatus.Specific.UpperSwitchAreaError                            // Upper jam error is active
	                AND #ix_PECFreUp                                                       // Upper jam sensor is free
	            THEN

	                #sUDT_HMIStatus.Specific.UpperSwitchAreaError := FALSE;                 // reset error

	            END_IF;

	            IF #sUDT_HMIStatus.Specific.LowerSwitchAreaError                            // lower jam error is active
	                AND #ix_PECFreDwn                                                     // Lower jam sensor is free
	            THEN

	                #sUDT_HMIStatus.Specific.LowerSwitchAreaError := FALSE;                 // reset error

	            END_IF;

	            #sUDT_HMIStatus.Specific.SwitchingTimerError := False;
	            #sUDT_HMIStatus.Specific.LimitSensorLowerPosition := False;
	            #sUDT_HMIStatus.Specific.LimitSensorUpperPosition := False;

	        END_IF;

	    END_REGION

	    REGION 2.2 - Set errors

	        // Upper Jam sensor blocked in movement
	        IF NOT #ix_PECFreUp AND #ss_ABSwitch_Interface.Positioning

	        THEN
	            #sUDT_HMIStatus.Specific.UpperSwitchAreaError := TRUE;                      // Set error upper jam sensor
	        END_IF;

	        // Lower Jam sensor blocked in movement
	        IF NOT #ix_PECFreDwn AND #ss_ABSwitch_Interface.Positioning
	        THEN
	            #sUDT_HMIStatus.Specific.LowerSwitchAreaError := TRUE;                      // Set error lower jam sensor
	        END_IF;

	        //Configuration error
	        #sx_ConfigurationError := (#iUDT_ABSwitchConfig.BrakingSpeedSetpoint > #iUDT_ABSwitchConfig.NominalSpeedSetPoint)
	        OR #iUDT_ABSwitchConfig.NominalSpeedSetPoint = 0
	        OR #iUDT_ABSwitchConfig.BrakingSpeedSetpoint = 0
	        OR #iUDT_ABSwitchConfig.ManualModeSpeed = 0
	        OR #iUDT_ABSwitchConfig.SwitchingTime = 0
	        OR #iUDT_ABSwitchConfig.JogNoHornTime = 0
	        OR (#iUDT_ABSwitchConfig.BrakingSpeedSetpoint > 500);

	        //Switching Time
	        #SwitchingTime(iudi_OnDelayTime := #iUDT_ABSwitchConfig.SwitchingTime,
	                       iudi_OffDelayTime := 0,
	                       ix_SignalToDelay := #sx_SemiAutomatic AND NOT #iqUDT_EquipmentControl.Request.SignalingRequest AND (#sx_UpRequest AND #ix_PRXUp) OR (#sx_DownRequest AND #ix_PRXDown));

	        IF #SwitchingTime.qx_DelayedSignal THEN
	            #sUDT_HMIStatus.Specific.SwitchingTimerError := True;
	        END_IF;

	        // Reference error - set error when more like one position sensor is active
	        #ti_ActiveSensor := 0;

	        //Position sensor up
	        IF NOT #ix_PRXUp THEN
	            #ti_ActiveSensor += 1;
	        END_IF;

	        //Position sensor down
	        IF NOT #ix_PRXDown THEN
	            #ti_ActiveSensor += 1;
	        END_IF;

	        //Brake sensor up
	        IF NOT #ix_PRXBrkUp THEN
	            #ti_ActiveSensor += 1;
	        END_IF;

	        //Brak sensor down
	        IF NOT #ix_PRXBrkDwn THEN
	            #ti_ActiveSensor += 1;
	        END_IF;

	        //Limit switch up
	        IF NOT #ix_LSUp THEN
	            #ti_ActiveSensor += 1;
	        END_IF;

	        //Limit switch down
	        IF NOT #ix_LSDwn THEN
	            #ti_ActiveSensor += 1;
	        END_IF;

	        IF #ti_ActiveSensor >= 2 THEN
	            #sUDT_HMIStatus.Specific.ReferenceError := True;
	        ELSE
	            #sUDT_HMIStatus.Specific.ReferenceError := False;
	        END_IF;

	        //Limit switch active
	        IF NOT #ix_LSUp THEN

	            #sUDT_HMIStatus.Specific.LimitSensorUpperPosition := True;

	        END_IF;

	        IF NOT #ix_LSDwn THEN

	            #sUDT_HMIStatus.Specific.LimitSensorLowerPosition := True;

	        END_IF;

	    END_REGION

	    REGION 2.3 - Common Error

	        #sUDT_Status.Error :=
	        #iqUDT_ABSwitchInterface.InternalErrorTracking                                 // or the AB switch conveyor detected an error in tracking
	        OR #iqUDT_ABSwitchInterface.InternalErrorVFD                                   // or there are errors in the VFD
	        OR NOT #ix_HardwareOk                                                               // or an internal error in the RIO panel occured
	        OR #sUDT_HMIStatus.Specific.UpperSwitchAreaError                                // or Upper jam PEC detected WHILE going Up
	        OR #sUDT_HMIStatus.Specific.LowerSwitchAreaError;                                // or Lower jam PEC detected while going Down

	    END_REGION

	END_REGION

	REGION 3 - Check conditions to set Equipment ready

	    //Conditions to set bit sx_Ready to operate
	    #sx_Ready := NOT #sUDT_Status.Error                                                // Error not present
	    AND #ix_SafetyOk                                                                  // Safety signalling OK
	    AND NOT #sUDT_HMIStatus.Specific.LimitSensorUpperPosition
	    AND NOT #sUDT_HMIStatus.Specific.LimitSensorLowerPosition;


	END_REGION

	REGION 4 - Stop Equipment

	    IF (#ix_SSMan                                                        // Manual mode is active
	        AND #sx_SemiAutomatic                                                       // AB switch is in semi-automatic mode
	        OR (NOT #iqUDT_EquipmentControl.Command.AutomaticOn                        // AB switch stops if the bit AutomaticOn from control block is false
	        AND NOT #ix_SSMan)                                               // Manual mode active bit
	        OR (NOT #sx_Ready                                                           // Bit AB switch ready to run in automatic mode
	        AND NOT #ix_SSMan)                                               // Manual mode active
	        OR #ix_SSMan                                                      // LCP is not set to automatic
	        OR NOT #ix_SafetyOk)                                                        // Safety is not ok
	    THEN                                                                            // Order to stop
	        #sx_Stopping := TRUE;                                                       // stopping is activated
	        #sx_SemiAutomatic := FALSE;                                                 // switch of automatic activ
	        #sx_StartReceived := FALSE;                                                 // Start command received from system

	    END_IF;

	    IF (#sx_Stopping                                                                 // stopping is activated
	        AND NOT #ss_ABSwitch_Interface.Positioning)                                       // The positioning device is not active positioning
	        OR NOT #sx_Ready                                                             // AB switch is not ready to run
	    THEN
	        #sx_Stopping := FALSE;                                                       // stopping is activated
	    END_IF;

	END_REGION

	REGION 5 - Start Semi-automatic mode

	    REGION 5.1 - Start

	        // if start (OS) is received from system, this is memorised until started in cascade
	        IF #iqUDT_EquipmentControl.Command.Start                                       // Start from system
	            AND #sx_Ready                                                               // Equipment has no errors
	        THEN
	            #sx_StartReceived := TRUE;                                                  // Start command received from system
	        END_IF;

	        IF #sx_StartReceived                                                            // Start command received from system
	            AND NOT #ix_SSMan                                                         // and the LCP is set to auto
	        THEN
	            #sx_SemiAutomatic := TRUE;                                                  // Automatic activated
	            #sx_StartReceived := FALSE;                                                 // Start command received from system
	        END_IF;

	    END_REGION

	END_REGION

	REGION 6 - Manual mode

	    REGION 6.1 - Jog signals

	        #sx_CombinedJogUp := #ix_SSMan                                                          // box in manual
	        AND #ix_PBUp;                                                                // If selected jog in positive direction

	        #sx_CombinedJogDown := #ix_SSMan                                                           // box in manual
	        AND #ix_PBDwn;                                                               // If selected jog in negative direction

	        // Detecting rising edge on manual jog Up
	        #R_TRIG_ManualJogUp(CLK := #sx_CombinedJogUp);

	        // Detecting rising edge on manual jog Down
	        #R_TRIG_ManualJogDown(CLK := #sx_CombinedJogDown);

	    END_REGION

	    REGION 6.2 - Manual PreStart up or down

	        // Pre start conditions to run in manual mode
	        #sx_PreStartManual := #ix_SSMan                                      // Manual mode active bit
	        AND #ix_SafetyOk                                                                // Safety healthy bit
	        AND NOT #iqUDT_ABSwitchInterface.InternalErrorVFD;                             // Profinet comunication or PN_DEvice not ok


	        IF #sx_PreStartManual                                                           // Pre start conditions to run in manual mode
	            AND (#R_TRIG_ManualJogUp.Q                                                  // Trigger to start AB switch run in manual jog mode UP
	            OR #R_TRIG_ManualJogDown.Q)                                                 // Trigger to start AB switch run in manual jog mode Down
	            AND NOT #Jog_Enable.qx_DelayedSignal
	        THEN

	            #iqUDT_EquipmentControl.Request.SignalingRequest := TRUE;                  // Request signaling TO control block before AB switch runs in manual mode

	        END_IF;

	    END_REGION

	    REGION 6.3 - Jog mode Up / Down

	        IF #sx_PreStartManual                                                           // IF in manual jog mode
	            AND (NOT #iqUDT_EquipmentControl.Request.SignalingRequest                  // Signaling request done
	            OR #Jog_Enable.qx_DelayedSignal)
	            AND #sx_CombinedJogUp                                                       // If selected jog in positive direction
	            AND NOT #sx_CombinedJogDown                                                 // And not selected jog in negative direction
	        THEN

	            #sx_JogUp := TRUE;                                                          // set jog positive
	            #sx_JogDown := FALSE;                                                       // reset jog negative
	            #sx_Jog := true;

	        ELSIF
	            #sx_PreStartManual                                                          // IF in manual jog mode
	            AND (NOT #iqUDT_EquipmentControl.Request.SignalingRequest                  // Signaling request done
	            OR #Jog_Enable.qx_DelayedSignal)
	            AND NOT #sx_CombinedJogUp                                                   // If selected jog in positive direction
	            AND #sx_CombinedJogDown                                                     // and there is command to jog in negative direction
	        THEN

	            #sx_JogUp := FALSE;                                                         // reset jog positive
	            #sx_JogDown := TRUE;                                                        // set jog negative
	            #sx_Jog := true;

	        ELSIF
	            NOT #sx_PreStartManual                                                      // If not in manual mode
	            OR (#sx_PreStartManual                                                      // or in manual mode
	            AND (#sx_CombinedJogUp                                                      // and jog positive is off
	            AND #sx_CombinedJogDown)                                                    // AND jog negative is off
	            OR (NOT #sx_CombinedJogUp                                                   // or jog positive is on
	            AND NOT #sx_CombinedJogDown))                                               // and jog negative is on
	        THEN

	            #sx_JogUp := FALSE;                                                         // reset jog positive
	            #sx_JogDown := FALSE;                                                       // reset jog negative
	            #sx_Jog := False;
	        END_IF;
	    END_REGION

	END_REGION

	REGION 7 - Automatic mode

	    REGION 7.1 - Semi automatic

	        IF #sx_SemiAutomatic                                                            // Not running Semi-Automatic
	            AND (#ii_Mode = #ci_UpperPosition
	            AND #ix_ChangeModeSignal)
	        THEN

	            #sx_PreStartSemiAutomaticUp := TRUE;

	            #sx_DownRequest := FALSE;                                                   // Reset down command
	            #sx_UpRequest := TRUE;                                                      // Set up command
	        END_IF;

	        IF #sx_SemiAutomatic                                                            // Not running Semi-Automatic
	            AND (#ii_Mode = #ci_LowerPosition
	            AND #ix_ChangeModeSignal)

	        THEN

	            #sx_PreStartSemiAutomaticDown := TRUE;

	            #sx_DownRequest := TRUE;                                                    // Reset down command
	            #sx_UpRequest := FALSE;                                                     // Set up command
	        END_IF;

	        #R_TRIG_PreStartSemiAutomaticUp(CLK := #sx_PreStartSemiAutomaticUp);
	        #R_TRIG_PreStartSemiAutomaticDown(CLK := #sx_PreStartSemiAutomaticDown);

